// eDataMappingVarNames.powermonitor_events_b_EL3443Warning: 				st_Variable:= IotExtractType(monitor.powermonitor.events.b_EL3443Warning, 0, 0); 
// eDataMappingVarNames.powermonitor_events_b_EL3443Error: 				st_Variable:= IotExtractType(monitor.powermonitor.events.b_EL3443Error, 0, 0); 
// eDataMappingVarNames.powermonitor_events_b_ACdirectionDataInvalid: 				st_Variable:= IotExtractType(monitor.powermonitor.events.b_ACdirectionDataInvalid, 0, 0); 
// eDataMappingVarNames.ACswitchgear_b_InputSectionAvailable: 				st_Variable:= IotExtractType(monitor.ACswitchgear.b_InputSectionAvailable, 0, 0); 
// eDataMappingVarNames.ACswitchgear_b_InputMCCBfb: 				st_Variable:= IotExtractType(monitor.ACswitchgear.b_InputMCCBfb, 0, 0); 
// eDataMappingVarNames.ACswitchgear_b_InputMCCBShuntOK: 				st_Variable:= IotExtractType(monitor.ACswitchgear.b_InputMCCBShuntOK, 0, 0); 
// eDataMappingVarNames.ACswitchgear_b_OutputMCCBfb: 				st_Variable:= IotExtractType(monitor.ACswitchgear.b_OutputMCCBfb, 0, 0); 
// eDataMappingVarNames.ACswitchgear_b_OutputMCCBShuntOK: 				st_Variable:= IotExtractType(monitor.ACswitchgear.b_OutputMCCBShuntOK, 0, 0); 
// eDataMappingVarNames.ACswitchgear_b_CEEprefuseOK: 				st_Variable:= IotExtractType(monitor.ACswitchgear.b_CEEprefuseOK, 0, 0); 
// eDataMappingVarNames.ACswitchgear_b_InputSynchronizerfb: 				st_Variable:= IotExtractType(monitor.ACswitchgear.b_InputSynchronizerfb, 0, 0); 
// eDataMappingVarNames.ACswitchgear_b_InputContactorfb: 				st_Variable:= IotExtractType(monitor.ACswitchgear.b_InputContactorfb, 0, 0); 
// eDataMappingVarNames.ACswitchgear_b_PENlinkfb: 				st_Variable:= IotExtractType(monitor.ACswitchgear.b_PENlinkfb, 0, 0); 
// eDataMappingVarNames.ACswitchgear_events_b_InputMCCBShuntFault: 				st_Variable:= IotExtractType(monitor.ACswitchgear.events.b_InputMCCBShuntFault, 0, 0); 
// eDataMappingVarNames.ACswitchgear_events_b_OutputMCCBShuntFault: 				st_Variable:= IotExtractType(monitor.ACswitchgear.events.b_OutputMCCBShuntFault, 0, 0); 
// eDataMappingVarNames.ACswitchgear_events_b_CEEprefuseFault: 				st_Variable:= IotExtractType(monitor.ACswitchgear.events.b_CEEprefuseFault, 0, 0); 
// eDataMappingVarNames.ACswitchgear_events_b_InputContactorFault: 				st_Variable:= IotExtractType(monitor.ACswitchgear.events.b_InputContactorFault, 0, 0); 
// eDataMappingVarNames.neutraltransformer_b_active: 				st_Variable:= IotExtractType(monitor.neutraltransformer.b_active, 0, 0); 
// eDataMappingVarNames.neutraltransformer_r_TemperaturePhase_0: 				st_Variable:= IotExtractType(monitor.neutraltransformer.r_TemperaturePhase[0], 1, 0); 
// eDataMappingVarNames.neutraltransformer_r_TemperaturePhase_1: 				st_Variable:= IotExtractType(monitor.neutraltransformer.r_TemperaturePhase[1], 1, 0); 
// eDataMappingVarNames.neutraltransformer_r_TemperaturePhase_2: 				st_Variable:= IotExtractType(monitor.neutraltransformer.r_TemperaturePhase[2], 1, 0); 
// eDataMappingVarNames.neutraltransformer_r_TemperaturePhase_3: 				st_Variable:= IotExtractType(monitor.neutraltransformer.r_TemperaturePhase[3], 1, 0); 
// eDataMappingVarNames.neutraltransformer_r_TemperaturePhase_4: 				st_Variable:= IotExtractType(monitor.neutraltransformer.r_TemperaturePhase[4], 1, 0); 
// eDataMappingVarNames.neutraltransformer_r_TemperaturePhase_5: 				st_Variable:= IotExtractType(monitor.neutraltransformer.r_TemperaturePhase[5], 1, 0); 
// eDataMappingVarNames.neutraltransformer_r_TemperaturePhase_6: 				st_Variable:= IotExtractType(monitor.neutraltransformer.r_TemperaturePhase[6], 1, 0); 
// eDataMappingVarNames.neutraltransformer_r_Powerload: 				st_Variable:= IotExtractType(monitor.neutraltransformer.r_Powerload, 1, 0); 
// eDataMappingVarNames.neutraltransformer_r_ratedPower: 				st_Variable:= IotExtractType(monitor.neutraltransformer.r_ratedPower, 0, 0); 
// eDataMappingVarNames.neutraltransformer_events_b_TemperatureHighPhase_1: 				st_Variable:= IotExtractType(monitor.neutraltransformer.events.b_TemperatureHighPhase[1], 0, 0); 
// eDataMappingVarNames.neutraltransformer_events_b_TemperatureHighPhase_2: 				st_Variable:= IotExtractType(monitor.neutraltransformer.events.b_TemperatureHighPhase[2], 0, 0); 
// eDataMappingVarNames.neutraltransformer_events_b_TemperatureHighPhase_3: 				st_Variable:= IotExtractType(monitor.neutraltransformer.events.b_TemperatureHighPhase[3], 0, 0); 
// eDataMappingVarNames.neutraltransformer_events_b_TemperatureTooHighPhase_1: 				st_Variable:= IotExtractType(monitor.neutraltransformer.events.b_TemperatureTooHighPhase[1], 0, 0); 
// eDataMappingVarNames.neutraltransformer_events_b_TemperatureTooHighPhase_2: 				st_Variable:= IotExtractType(monitor.neutraltransformer.events.b_TemperatureTooHighPhase[2], 0, 0); 
// eDataMappingVarNames.neutraltransformer_events_b_TemperatureTooHighPhase_3: 				st_Variable:= IotExtractType(monitor.neutraltransformer.events.b_TemperatureTooHighPhase[3], 0, 0); 
// eDataMappingVarNames.neutraltransformer_events_b_VoltageUnbalanceHigh: 				st_Variable:= IotExtractType(monitor.neutraltransformer.events.b_VoltageUnbalanceHigh, 0, 0); 
// eDataMappingVarNames.neutraltransformer_events_b_VoltageUnbalanceTooHigh: 				st_Variable:= IotExtractType(monitor.neutraltransformer.events.b_VoltageUnbalanceTooHigh, 0, 0); 
// eDataMappingVarNames.neutraltransformer_events_b_NeutralCurrentHigh: 				st_Variable:= IotExtractType(monitor.neutraltransformer.events.b_NeutralCurrentHigh, 0, 0); 
// eDataMappingVarNames.neutraltransformer_events_b_NeutralCurrentTooHigh: 				st_Variable:= IotExtractType(monitor.neutraltransformer.events.b_NeutralCurrentTooHigh, 0, 0); 
// eDataMappingVarNames.neutraltransformer_events_b_OvercurrentWarning: 				st_Variable:= IotExtractType(monitor.neutraltransformer.events.b_OvercurrentWarning, 0, 0); 
// eDataMappingVarNames.neutraltransformer_events_b_OvercurrentAlarm: 				st_Variable:= IotExtractType(monitor.neutraltransformer.events.b_OvercurrentAlarm, 0, 0); 
// eDataMappingVarNames.DCswitchgear_b_CouplingState: 				st_Variable:= IotExtractType(monitor.DCswitchgear.b_CouplingState, 0, 0); 
// eDataMappingVarNames.DCswitchgear_r_Current: 				st_Variable:= IotExtractType(monitor.DCswitchgear.r_Current, 0, 0); 
// eDataMappingVarNames.DCswitchgear_r_ratedCurrent: 				st_Variable:= IotExtractType(monitor.DCswitchgear.r_ratedCurrent, 0, 0); 
// eDataMappingVarNames.battery_BatteryInfo_b_BMSHeartBeatOK: 				st_Variable:= IotExtractType(monitor.battery.BatteryInfo.b_BMSHeartBeatOK, 0, 0); 
// eDataMappingVarNames.battery_BatteryInfo_e_BMS_PowerOnStatus: 				st_Variable:= IotExtractType(monitor.battery.BatteryInfo.e_BMS_PowerOnStatus, 0, 0); 
// eDataMappingVarNames.battery_BatteryInfo_e_BMS_Status: 				st_Variable:= IotExtractType(monitor.battery.BatteryInfo.e_BMS_Status, 0, 0); 
// eDataMappingVarNames.battery_BatteryInfo_r_SystemVoltage: 				st_Variable:= IotExtractType(monitor.battery.BatteryInfo.r_SystemVoltage, 1, 0); 
// eDataMappingVarNames.battery_BatteryInfo_r_SystemCurrent: 				st_Variable:= IotExtractType(monitor.battery.BatteryInfo.r_SystemCurrent, 1, 0); 
// eDataMappingVarNames.battery_BatteryInfo_r_SOC: 				st_Variable:= IotExtractType(monitor.battery.BatteryInfo.r_SOC, 1, 0); 
// eDataMappingVarNames.battery_BatteryInfo_r_SOH: 				st_Variable:= IotExtractType(monitor.battery.BatteryInfo.r_SOH, 1, 0); 
// eDataMappingVarNames.battery_BatteryInfo_ar_CellVoltage_0: 				st_Variable:= IotExtractType(monitor.battery.BatteryInfo.ar_CellVoltage[0], 2, 0); 
// eDataMappingVarNames.battery_BatteryInfo_ar_CellVoltage_1: 				st_Variable:= IotExtractType(monitor.battery.BatteryInfo.ar_CellVoltage[1], 2, 0); 
// eDataMappingVarNames.battery_BatteryInfo_ar_CellVoltage_2: 				st_Variable:= IotExtractType(monitor.battery.BatteryInfo.ar_CellVoltage[2], 2, 0); 
// eDataMappingVarNames.battery_BatteryInfo_ar_CellTemperature_0: 				st_Variable:= IotExtractType(monitor.battery.BatteryInfo.ar_CellTemperature[0], 1, 0); 
// eDataMappingVarNames.battery_BatteryInfo_ar_CellTemperature_1: 				st_Variable:= IotExtractType(monitor.battery.BatteryInfo.ar_CellTemperature[1], 1, 0); 
// eDataMappingVarNames.battery_BatteryInfo_ar_CellTemperature_2: 				st_Variable:= IotExtractType(monitor.battery.BatteryInfo.ar_CellTemperature[2], 1, 0); 
// eDataMappingVarNames.battery_BatteryInfo_r_MaxChargeCurrentAllowed: 				st_Variable:= IotExtractType(monitor.battery.BatteryInfo.r_MaxChargeCurrentAllowed, 0, 0); 
// eDataMappingVarNames.battery_BatteryInfo_r_MaxDischargeCurrentAllowed: 				st_Variable:= IotExtractType(monitor.battery.BatteryInfo.r_MaxDischargeCurrentAllowed, 0, 0); 
// eDataMappingVarNames.battery_BatteryInfo_r_MaxChargePowerAllowed: 				st_Variable:= IotExtractType(monitor.battery.BatteryInfo.r_MaxChargePowerAllowed, 0, 0); 
// eDataMappingVarNames.battery_BatteryInfo_r_MaxDischargePowerAllowed: 				st_Variable:= IotExtractType(monitor.battery.BatteryInfo.r_MaxDischargePowerAllowed, 0, 0); 
// eDataMappingVarNames.battery_BatteryInfo_r_MaxSystemVoltageAllowed: 				st_Variable:= IotExtractType(monitor.battery.BatteryInfo.r_MaxSystemVoltageAllowed, 0, 0); 
// eDataMappingVarNames.battery_BatteryInfo_r_MinSystemVoltageAllowed: 				st_Variable:= IotExtractType(monitor.battery.BatteryInfo.r_MinSystemVoltageAllowed, 0, 0); 
// eDataMappingVarNames.battery_BatteryInfo_r_SystemPower: 				st_Variable:= IotExtractType(monitor.battery.BatteryInfo.r_SystemPower, 1, 0); 
// eDataMappingVarNames.battery_BatteryInfo_r_ChargeSOE: 				st_Variable:= IotExtractType(monitor.battery.BatteryInfo.r_ChargeSOE, 0, 0); 
// eDataMappingVarNames.battery_BatteryInfo_r_DischargeSOE: 				st_Variable:= IotExtractType(monitor.battery.BatteryInfo.r_DischargeSOE, 0, 0); 
// eDataMappingVarNames.battery_BatteryInfo_r_RemainingChargeEnergy: 				st_Variable:= IotExtractType(monitor.battery.BatteryInfo.r_RemainingChargeEnergy, 0, 0); 
// eDataMappingVarNames.battery_BatteryInfo_r_RemainingDischargeEnergy: 				st_Variable:= IotExtractType(monitor.battery.BatteryInfo.r_RemainingDischargeEnergy, 0, 0); 
// eDataMappingVarNames.battery_BatteryInfo_r_HistAccChargeEnergy: 				st_Variable:= IotExtractType(monitor.battery.BatteryInfo.r_HistAccChargeEnergy, 0, 0); 
// eDataMappingVarNames.battery_BatteryInfo_r_HistAccDischargeEnergy: 				st_Variable:= IotExtractType(monitor.battery.BatteryInfo.r_HistAccDischargeEnergy, 0, 0); 
// eDataMappingVarNames.battery_BatteryInfo_r_ratedPower: 				st_Variable:= IotExtractType(monitor.battery.BatteryInfo.r_ratedPower, 0, 0); 
// eDataMappingVarNames.battery_BatteryInfo_r_ratedCurrent: 				st_Variable:= IotExtractType(monitor.battery.BatteryInfo.r_ratedCurrent, 0, 0); 
// eDataMappingVarNames.battery_BatteryInfo_r_ratedEnergyCapacity: 				st_Variable:= IotExtractType(monitor.battery.BatteryInfo.r_ratedEnergyCapacity, 0, 0); 
// eDataMappingVarNames.battery_BatteryInfo_ui_CycleCount: 				st_Variable:= IotExtractType(monitor.battery.BatteryInfo.ui_CycleCount, 0, 0); 
// eDataMappingVarNames.battery_BatteryInfo_r_SOCScaled: 				st_Variable:= IotExtractType(monitor.battery.BatteryInfo.r_SOCScaled, 1, 0); 
// eDataMappingVarNames.battery_BatteryInfo_b_chargingAllowed: 				st_Variable:= IotExtractType(monitor.battery.BatteryInfo.b_chargingAllowed, 0, 0); 
// eDataMappingVarNames.battery_BatteryInfo_b_dischargingAllowed: 				st_Variable:= IotExtractType(monitor.battery.BatteryInfo.b_dischargingAllowed, 0, 0); 
// eDataMappingVarNames.battery_BatteryInfo_r_RemainingDischargeEnergyNett: 				st_Variable:= IotExtractType(monitor.battery.BatteryInfo.r_RemainingDischargeEnergyNett, 0, 0); 
// eDataMappingVarNames.battery_BatteryInfo_r_RemainingChargeEnergyNett: 				st_Variable:= IotExtractType(monitor.battery.BatteryInfo.r_RemainingChargeEnergyNett, 0, 0); 
// eDataMappingVarNames.battery_BatteryInfo_r_maxVoltageEver: 				st_Variable:= IotExtractType(monitor.battery.BatteryInfo.r_maxVoltageEver, 1, 0); 
// eDataMappingVarNames.battery_BatteryInfo_r_maxChargeCurrentEver: 				st_Variable:= IotExtractType(monitor.battery.BatteryInfo.r_maxChargeCurrentEver, 1, 0); 
// eDataMappingVarNames.battery_BatteryInfo_r_maxDischargeCurrentEver: 				st_Variable:= IotExtractType(monitor.battery.BatteryInfo.r_maxDischargeCurrentEver, 1, 0); 
// eDataMappingVarNames.battery_T_RemainingTimeToAutoCalibration: 				st_Variable:= IotExtractType(monitor.battery.T_RemainingTimeToAutoCalibration, 0, 0); 
// eDataMappingVarNames.battery_MBMU_GeneralSBMUStatus_0: 				st_Variable:= IotExtractType(monitor.battery.MBMU.GeneralSBMUStatus[0], 0, 0); 
// eDataMappingVarNames.battery_MBMU_GeneralSBMUStatus_1: 				st_Variable:= IotExtractType(monitor.battery.MBMU.GeneralSBMUStatus[1], 0, 0); 
// eDataMappingVarNames.battery_MBMU_GeneralSBMUStatus_2: 				st_Variable:= IotExtractType(monitor.battery.MBMU.GeneralSBMUStatus[2], 0, 0); 
// eDataMappingVarNames.battery_MBMU_GeneralSBMUStatus_3: 				st_Variable:= IotExtractType(monitor.battery.MBMU.GeneralSBMUStatus[3], 0, 0); 
// eDataMappingVarNames.battery_MBMU_GeneralSBMUStatus_4: 				st_Variable:= IotExtractType(monitor.battery.MBMU.GeneralSBMUStatus[4], 0, 0); 
// eDataMappingVarNames.battery_MBMU_GeneralSBMUStatus_5: 				st_Variable:= IotExtractType(monitor.battery.MBMU.GeneralSBMUStatus[5], 0, 0); 
// eDataMappingVarNames.battery_MBMU_GeneralSBMUStatus_6: 				st_Variable:= IotExtractType(monitor.battery.MBMU.GeneralSBMUStatus[6], 0, 0); 
// eDataMappingVarNames.battery_MBMU_GeneralSBMUStatus_7: 				st_Variable:= IotExtractType(monitor.battery.MBMU.GeneralSBMUStatus[7], 0, 0); 
// eDataMappingVarNames.battery_MBMU_GeneralSBMUStatus_8: 				st_Variable:= IotExtractType(monitor.battery.MBMU.GeneralSBMUStatus[8], 0, 0); 
// eDataMappingVarNames.battery_MBMU_GeneralSBMUStatus_9: 				st_Variable:= IotExtractType(monitor.battery.MBMU.GeneralSBMUStatus[9], 0, 0); 
// eDataMappingVarNames.battery_MBMU_GeneralSBMUStatus_10: 				st_Variable:= IotExtractType(monitor.battery.MBMU.GeneralSBMUStatus[10], 0, 0); 
// eDataMappingVarNames.battery_MBMU_GeneralSBMUStatus_11: 				st_Variable:= IotExtractType(monitor.battery.MBMU.GeneralSBMUStatus[11], 0, 0); 
// eDataMappingVarNames.battery_MBMU_GeneralSBMUStatus_12: 				st_Variable:= IotExtractType(monitor.battery.MBMU.GeneralSBMUStatus[12], 0, 0); 
// eDataMappingVarNames.battery_MBMU_GeneralSBMUStatus_13: 				st_Variable:= IotExtractType(monitor.battery.MBMU.GeneralSBMUStatus[13], 0, 0); 
// eDataMappingVarNames.battery_MBMU_GeneralSBMUStatus_14: 				st_Variable:= IotExtractType(monitor.battery.MBMU.GeneralSBMUStatus[14], 0, 0); 
// eDataMappingVarNames.battery_MBMU_GeneralSBMUStatus_15: 				st_Variable:= IotExtractType(monitor.battery.MBMU.GeneralSBMUStatus[15], 0, 0); 
// eDataMappingVarNames.battery_MBMU_MBMUStatus_0: 				st_Variable:= IotExtractType(monitor.battery.MBMU.MBMUStatus[0], 0, 0); 
// eDataMappingVarNames.battery_MBMU_MBMUStatus_1: 				st_Variable:= IotExtractType(monitor.battery.MBMU.MBMUStatus[1], 0, 0); 
// eDataMappingVarNames.battery_MBMU_MBMUStatus_2: 				st_Variable:= IotExtractType(monitor.battery.MBMU.MBMUStatus[2], 0, 0); 
// eDataMappingVarNames.battery_MBMU_MBMUStatus_3: 				st_Variable:= IotExtractType(monitor.battery.MBMU.MBMUStatus[3], 0, 0); 
// eDataMappingVarNames.battery_MBMU_MBMUStatus_4: 				st_Variable:= IotExtractType(monitor.battery.MBMU.MBMUStatus[4], 0, 0); 
// eDataMappingVarNames.battery_MBMU_MBMUStatus_5: 				st_Variable:= IotExtractType(monitor.battery.MBMU.MBMUStatus[5], 0, 0); 
// eDataMappingVarNames.battery_MBMU_MBMUStatus_6: 				st_Variable:= IotExtractType(monitor.battery.MBMU.MBMUStatus[6], 0, 0); 
// eDataMappingVarNames.battery_MBMU_MBMUStatus_7: 				st_Variable:= IotExtractType(monitor.battery.MBMU.MBMUStatus[7], 0, 0); 
// eDataMappingVarNames.battery_MBMU_MBMUStatus_8: 				st_Variable:= IotExtractType(monitor.battery.MBMU.MBMUStatus[8], 0, 0); 
// eDataMappingVarNames.battery_MBMU_MBMUStatus_9: 				st_Variable:= IotExtractType(monitor.battery.MBMU.MBMUStatus[9], 0, 0); 
// eDataMappingVarNames.battery_MBMU_MBMUStatus_10: 				st_Variable:= IotExtractType(monitor.battery.MBMU.MBMUStatus[10], 0, 0); 
// eDataMappingVarNames.battery_MBMU_MBMUStatus_11: 				st_Variable:= IotExtractType(monitor.battery.MBMU.MBMUStatus[11], 0, 0); 
// eDataMappingVarNames.battery_MBMU_MBMUStatus_12: 				st_Variable:= IotExtractType(monitor.battery.MBMU.MBMUStatus[12], 0, 0); 
// eDataMappingVarNames.battery_MBMU_MBMUStatus_13: 				st_Variable:= IotExtractType(monitor.battery.MBMU.MBMUStatus[13], 0, 0); 
// eDataMappingVarNames.battery_MBMU_MBMUStatus_14: 				st_Variable:= IotExtractType(monitor.battery.MBMU.MBMUStatus[14], 0, 0); 
// eDataMappingVarNames.battery_MBMU_MBMUStatus_15: 				st_Variable:= IotExtractType(monitor.battery.MBMU.MBMUStatus[15], 0, 0); 
// eDataMappingVarNames.battery_MBMU_s_MBMU_SWVer: 				st_Variable:= IotExtractType(monitor.battery.MBMU.s_MBMU_SWVer, 0, 0); 
// eDataMappingVarNames.battery_MBMU_s_MBMU_HWVer: 				st_Variable:= IotExtractType(monitor.battery.MBMU.s_MBMU_HWVer, 0, 0); 
// eDataMappingVarNames.battery_MBMU_s_ETH_SWVer: 				st_Variable:= IotExtractType(monitor.battery.MBMU.s_ETH_SWVer, 0, 0); 
// eDataMappingVarNames.battery_MBMU_r_ETH_HWVer: 				st_Variable:= IotExtractType(monitor.battery.MBMU.r_ETH_HWVer, 0, 0); 
// eDataMappingVarNames.battery_MBMU_by_NumberOfSubSystems: 				st_Variable:= IotExtractType(monitor.battery.MBMU.by_NumberOfSubSystems, 0, 0); 
// eDataMappingVarNames.battery_MBMU_DateTime_0: 				st_Variable:= IotExtractType(monitor.battery.MBMU.DateTime[0], 0, 0); 
// eDataMappingVarNames.battery_MBMU_DateTime_1: 				st_Variable:= IotExtractType(monitor.battery.MBMU.DateTime[1], 0, 0); 
// eDataMappingVarNames.battery_MBMU_DateTime_2: 				st_Variable:= IotExtractType(monitor.battery.MBMU.DateTime[2], 0, 0); 
// eDataMappingVarNames.battery_MBMU_DateTime_3: 				st_Variable:= IotExtractType(monitor.battery.MBMU.DateTime[3], 0, 0); 
// eDataMappingVarNames.battery_MBMU_DateTime_4: 				st_Variable:= IotExtractType(monitor.battery.MBMU.DateTime[4], 0, 0); 
// eDataMappingVarNames.battery_MBMU_DateTime_5: 				st_Variable:= IotExtractType(monitor.battery.MBMU.DateTime[5], 0, 0); 
// eDataMappingVarNames.battery_MBMU_b_InsulationSwitchOpen: 				st_Variable:= IotExtractType(monitor.battery.MBMU.b_InsulationSwitchOpen, 0, 0); 
// eDataMappingVarNames.battery_MBMU_BatteryStatus_b_BMSHeartBeatOK: 				st_Variable:= IotExtractType(monitor.battery.MBMU.BatteryStatus.b_BMSHeartBeatOK, 0, 0); 
// eDataMappingVarNames.battery_MBMU_BatteryStatus_e_BMS_PowerOnStatus: 				st_Variable:= IotExtractType(monitor.battery.MBMU.BatteryStatus.e_BMS_PowerOnStatus, 0, 0); 
// eDataMappingVarNames.battery_MBMU_BatteryStatus_e_BMS_Status: 					st_Variable:= IotExtractType(monitor.battery.MBMU.BatteryStatus.e_BMS_Status, 0, 0); 
// eDataMappingVarNames.battery_MBMU_BatteryStatus_r_SystemVoltage: 				st_Variable:= IotExtractType(monitor.battery.MBMU.BatteryStatus.r_SystemVoltage, 0, 0); 
// eDataMappingVarNames.battery_MBMU_BatteryStatus_r_SystemCurrent: 				st_Variable:= IotExtractType(monitor.battery.MBMU.BatteryStatus.r_SystemCurrent, 0, 0); 
// eDataMappingVarNames.battery_MBMU_BatteryStatus_r_SOC: 							st_Variable:= IotExtractType(monitor.battery.MBMU.BatteryStatus.r_SOC, 1, 0); 
// eDataMappingVarNames.battery_MBMU_BatteryStatus_r_SOH: 							st_Variable:= IotExtractType(monitor.battery.MBMU.BatteryStatus.r_SOH, 1, 0); 
// eDataMappingVarNames.battery_MBMU_BatteryStatus_ar_CellVoltage_0: 				st_Variable:= IotExtractType(monitor.battery.MBMU.BatteryStatus.ar_CellVoltage[0], 2, 0); 
// eDataMappingVarNames.battery_MBMU_BatteryStatus_ar_CellVoltage_1: 				st_Variable:= IotExtractType(monitor.battery.MBMU.BatteryStatus.ar_CellVoltage[1], 2, 0); 
// eDataMappingVarNames.battery_MBMU_BatteryStatus_ar_CellVoltage_2: 				st_Variable:= IotExtractType(monitor.battery.MBMU.BatteryStatus.ar_CellVoltage[2], 2, 0); 
// eDataMappingVarNames.battery_MBMU_BatteryStatus_ar_CellTemperature_0: 				st_Variable:= IotExtractType(monitor.battery.MBMU.BatteryStatus.ar_CellTemperature[0], 1, 0); 
// eDataMappingVarNames.battery_MBMU_BatteryStatus_ar_CellTemperature_1: 				st_Variable:= IotExtractType(monitor.battery.MBMU.BatteryStatus.ar_CellTemperature[1], 1, 0); 
// eDataMappingVarNames.battery_MBMU_BatteryStatus_ar_CellTemperature_2: 				st_Variable:= IotExtractType(monitor.battery.MBMU.BatteryStatus.ar_CellTemperature[2], 1, 0); 
// eDataMappingVarNames.battery_MBMU_BatteryStatus_r_MaxChargeCurrentAllowed: 				st_Variable:= IotExtractType(monitor.battery.MBMU.BatteryStatus.r_MaxChargeCurrentAllowed, 0, 0); 
// eDataMappingVarNames.battery_MBMU_BatteryStatus_r_MaxDischargeCurrentAllowed: 				st_Variable:= IotExtractType(monitor.battery.MBMU.BatteryStatus.r_MaxDischargeCurrentAllowed, 0, 0); 
// eDataMappingVarNames.battery_MBMU_BatteryStatus_r_MaxChargePowerAllowed: 				st_Variable:= IotExtractType(monitor.battery.MBMU.BatteryStatus.r_MaxChargePowerAllowed, 0, 0); 
// eDataMappingVarNames.battery_MBMU_BatteryStatus_r_MaxDischargePowerAllowed: 				st_Variable:= IotExtractType(monitor.battery.MBMU.BatteryStatus.r_MaxDischargePowerAllowed, 0, 0); 
// eDataMappingVarNames.battery_MBMU_BatteryStatus_r_MaxSystemVoltageAllowed: 				st_Variable:= IotExtractType(monitor.battery.MBMU.BatteryStatus.r_MaxSystemVoltageAllowed, 0, 0); 
// eDataMappingVarNames.battery_MBMU_BatteryStatus_r_MinSystemVoltageAllowed: 				st_Variable:= IotExtractType(monitor.battery.MBMU.BatteryStatus.r_MinSystemVoltageAllowed, 0, 0); 
// eDataMappingVarNames.battery_MBMU_BatteryStatus_r_SystemPower: 				st_Variable:= IotExtractType(monitor.battery.MBMU.BatteryStatus.r_SystemPower, 1, 0); 
// eDataMappingVarNames.battery_MBMU_BatteryStatus_r_ChargeSOE: 				st_Variable:= IotExtractType(monitor.battery.MBMU.BatteryStatus.r_ChargeSOE, 0, 0); 
// eDataMappingVarNames.battery_MBMU_BatteryStatus_r_DischargeSOE: 				st_Variable:= IotExtractType(monitor.battery.MBMU.BatteryStatus.r_DischargeSOE, 0, 0); 
// eDataMappingVarNames.battery_MBMU_BatteryStatus_r_RemainingChargeEnergy: 				st_Variable:= IotExtractType(monitor.battery.MBMU.BatteryStatus.r_RemainingChargeEnergy, 0, 0); 
// eDataMappingVarNames.battery_MBMU_BatteryStatus_r_RemainingDischargeEnergy: 				st_Variable:= IotExtractType(monitor.battery.MBMU.BatteryStatus.r_RemainingDischargeEnergy, 0, 0); 
// eDataMappingVarNames.battery_MBMU_BatteryStatus_r_HistAccChargeEnergy: 				st_Variable:= IotExtractType(monitor.battery.MBMU.BatteryStatus.r_HistAccChargeEnergy, 0, 0); 
// eDataMappingVarNames.battery_MBMU_BatteryStatus_r_HistAccDischargeEnergy: 				st_Variable:= IotExtractType(monitor.battery.MBMU.BatteryStatus.r_HistAccDischargeEnergy, 0, 0); 
// eDataMappingVarNames.battery_SBMU_0_w_SystemWarning: 				st_Variable:= IotExtractType(monitor.battery.SBMU[0].w_SystemWarning, 0, 0); 
// eDataMappingVarNames.battery_SBMU_1_w_SystemWarning: 				st_Variable:= IotExtractType(monitor.battery.SBMU[1].w_SystemWarning, 0, 0); 
// eDataMappingVarNames.battery_SBMU_2_w_SystemWarning: 				st_Variable:= IotExtractType(monitor.battery.SBMU[2].w_SystemWarning, 0, 0); 
// eDataMappingVarNames.battery_SBMU_3_w_SystemWarning: 				st_Variable:= IotExtractType(monitor.battery.SBMU[3].w_SystemWarning, 0, 0); 
// eDataMappingVarNames.battery_SBMU_0_SystemAlarm_0: 				st_Variable:= IotExtractType(monitor.battery.SBMU[0].SystemAlarm[0], 0, 0); 
// eDataMappingVarNames.battery_SBMU_1_SystemAlarm_0: 				st_Variable:= IotExtractType(monitor.battery.SBMU[1].SystemAlarm[0], 0, 0); 
// eDataMappingVarNames.battery_SBMU_2_SystemAlarm_0: 				st_Variable:= IotExtractType(monitor.battery.SBMU[2].SystemAlarm[0], 0, 0); 
// eDataMappingVarNames.battery_SBMU_3_SystemAlarm_0: 				st_Variable:= IotExtractType(monitor.battery.SBMU[3].SystemAlarm[0], 0, 0); 
// eDataMappingVarNames.battery_SBMU_0_SystemAlarm_1: 				st_Variable:= IotExtractType(monitor.battery.SBMU[0].SystemAlarm[1], 0, 0); 
// eDataMappingVarNames.battery_SBMU_1_SystemAlarm_1: 				st_Variable:= IotExtractType(monitor.battery.SBMU[1].SystemAlarm[1], 0, 0); 
// eDataMappingVarNames.battery_SBMU_2_SystemAlarm_1: 				st_Variable:= IotExtractType(monitor.battery.SBMU[2].SystemAlarm[1], 0, 0); 
// eDataMappingVarNames.battery_SBMU_3_SystemAlarm_1: 				st_Variable:= IotExtractType(monitor.battery.SBMU[3].SystemAlarm[1], 0, 0); 
// eDataMappingVarNames.battery_SBMU_0_SystemAlarm_2: 				st_Variable:= IotExtractType(monitor.battery.SBMU[0].SystemAlarm[2], 0, 0); 
// eDataMappingVarNames.battery_SBMU_1_SystemAlarm_2: 				st_Variable:= IotExtractType(monitor.battery.SBMU[1].SystemAlarm[2], 0, 0); 
// eDataMappingVarNames.battery_SBMU_2_SystemAlarm_2: 				st_Variable:= IotExtractType(monitor.battery.SBMU[2].SystemAlarm[2], 0, 0); 
// eDataMappingVarNames.battery_SBMU_3_SystemAlarm_2: 				st_Variable:= IotExtractType(monitor.battery.SBMU[3].SystemAlarm[2], 0, 0); 
// eDataMappingVarNames.battery_SBMU_0_b_PrechargeRelayClosed: 				st_Variable:= IotExtractType(monitor.battery.SBMU[0].b_PrechargeRelayClosed, 0, 0); 
// eDataMappingVarNames.battery_SBMU_1_b_PrechargeRelayClosed: 				st_Variable:= IotExtractType(monitor.battery.SBMU[1].b_PrechargeRelayClosed, 0, 0); 
// eDataMappingVarNames.battery_SBMU_2_b_PrechargeRelayClosed: 				st_Variable:= IotExtractType(monitor.battery.SBMU[2].b_PrechargeRelayClosed, 0, 0); 
// eDataMappingVarNames.battery_SBMU_3_b_PrechargeRelayClosed: 				st_Variable:= IotExtractType(monitor.battery.SBMU[3].b_PrechargeRelayClosed, 0, 0); 
// eDataMappingVarNames.battery_SBMU_0_b_MainPosRelayClosed: 				st_Variable:= IotExtractType(monitor.battery.SBMU[0].b_MainPosRelayClosed, 0, 0); 
// eDataMappingVarNames.battery_SBMU_1_b_MainPosRelayClosed: 				st_Variable:= IotExtractType(monitor.battery.SBMU[1].b_MainPosRelayClosed, 0, 0); 
// eDataMappingVarNames.battery_SBMU_2_b_MainPosRelayClosed: 				st_Variable:= IotExtractType(monitor.battery.SBMU[2].b_MainPosRelayClosed, 0, 0); 
// eDataMappingVarNames.battery_SBMU_3_b_MainPosRelayClosed: 				st_Variable:= IotExtractType(monitor.battery.SBMU[3].b_MainPosRelayClosed, 0, 0); 
// eDataMappingVarNames.battery_SBMU_0_b_MainNegRelayClosed: 				st_Variable:= IotExtractType(monitor.battery.SBMU[0].b_MainNegRelayClosed, 0, 0); 
// eDataMappingVarNames.battery_SBMU_1_b_MainNegRelayClosed: 				st_Variable:= IotExtractType(monitor.battery.SBMU[1].b_MainNegRelayClosed, 0, 0); 
// eDataMappingVarNames.battery_SBMU_2_b_MainNegRelayClosed: 				st_Variable:= IotExtractType(monitor.battery.SBMU[2].b_MainNegRelayClosed, 0, 0); 
// eDataMappingVarNames.battery_SBMU_3_b_MainNegRelayClosed: 				st_Variable:= IotExtractType(monitor.battery.SBMU[3].b_MainNegRelayClosed, 0, 0); 
// eDataMappingVarNames.battery_SBMU_0_b_ControlBoxFanOn: 				st_Variable:= IotExtractType(monitor.battery.SBMU[0].b_ControlBoxFanOn, 0, 0); 
// eDataMappingVarNames.battery_SBMU_1_b_ControlBoxFanOn: 				st_Variable:= IotExtractType(monitor.battery.SBMU[1].b_ControlBoxFanOn, 0, 0); 
// eDataMappingVarNames.battery_SBMU_2_b_ControlBoxFanOn: 				st_Variable:= IotExtractType(monitor.battery.SBMU[2].b_ControlBoxFanOn, 0, 0); 
// eDataMappingVarNames.battery_SBMU_3_b_ControlBoxFanOn: 				st_Variable:= IotExtractType(monitor.battery.SBMU[3].b_ControlBoxFanOn, 0, 0); 
// eDataMappingVarNames.battery_SBMU_0_b_BalanceStatus: 				st_Variable:= IotExtractType(monitor.battery.SBMU[0].b_BalanceStatus, 0, 0); 
// eDataMappingVarNames.battery_SBMU_1_b_BalanceStatus: 				st_Variable:= IotExtractType(monitor.battery.SBMU[1].b_BalanceStatus, 0, 0); 
// eDataMappingVarNames.battery_SBMU_2_b_BalanceStatus: 				st_Variable:= IotExtractType(monitor.battery.SBMU[2].b_BalanceStatus, 0, 0); 
// eDataMappingVarNames.battery_SBMU_3_b_BalanceStatus: 				st_Variable:= IotExtractType(monitor.battery.SBMU[3].b_BalanceStatus, 0, 0); 
// eDataMappingVarNames.battery_SBMU_0_b_DoorState: 				st_Variable:= IotExtractType(monitor.battery.SBMU[0].b_DoorState, 0, 0); 
// eDataMappingVarNames.battery_SBMU_1_b_DoorState: 				st_Variable:= IotExtractType(monitor.battery.SBMU[1].b_DoorState, 0, 0); 
// eDataMappingVarNames.battery_SBMU_2_b_DoorState: 				st_Variable:= IotExtractType(monitor.battery.SBMU[2].b_DoorState, 0, 0); 
// eDataMappingVarNames.battery_SBMU_3_b_DoorState: 				st_Variable:= IotExtractType(monitor.battery.SBMU[3].b_DoorState, 0, 0); 
// eDataMappingVarNames.battery_SBMU_0_s_SBMU_SWVer: 				st_Variable:= IotExtractType(monitor.battery.SBMU[0].s_SBMU_SWVer, 0, 0); 
// eDataMappingVarNames.battery_SBMU_1_s_SBMU_SWVer: 				st_Variable:= IotExtractType(monitor.battery.SBMU[1].s_SBMU_SWVer, 0, 0); 
// eDataMappingVarNames.battery_SBMU_2_s_SBMU_SWVer: 				st_Variable:= IotExtractType(monitor.battery.SBMU[2].s_SBMU_SWVer, 0, 0); 
// eDataMappingVarNames.battery_SBMU_3_s_SBMU_SWVer: 				st_Variable:= IotExtractType(monitor.battery.SBMU[3].s_SBMU_SWVer, 0, 0); 
// eDataMappingVarNames.battery_SBMU_0_s_SBMU_HWVer: 				st_Variable:= IotExtractType(monitor.battery.SBMU[0].s_SBMU_HWVer, 0, 0); 
// eDataMappingVarNames.battery_SBMU_1_s_SBMU_HWVer: 				st_Variable:= IotExtractType(monitor.battery.SBMU[1].s_SBMU_HWVer, 0, 0); 
// eDataMappingVarNames.battery_SBMU_2_s_SBMU_HWVer: 				st_Variable:= IotExtractType(monitor.battery.SBMU[2].s_SBMU_HWVer, 0, 0); 
// eDataMappingVarNames.battery_SBMU_3_s_SBMU_HWVer: 				st_Variable:= IotExtractType(monitor.battery.SBMU[3].s_SBMU_HWVer, 0, 0); 
// eDataMappingVarNames.battery_SBMU_0_s_CSC_SWVer: 				st_Variable:= IotExtractType(monitor.battery.SBMU[0].s_CSC_SWVer, 0, 0); 
// eDataMappingVarNames.battery_SBMU_1_s_CSC_SWVer: 				st_Variable:= IotExtractType(monitor.battery.SBMU[1].s_CSC_SWVer, 0, 0); 
// eDataMappingVarNames.battery_SBMU_2_s_CSC_SWVer: 				st_Variable:= IotExtractType(monitor.battery.SBMU[2].s_CSC_SWVer, 0, 0); 
// eDataMappingVarNames.battery_SBMU_3_s_CSC_SWVer: 				st_Variable:= IotExtractType(monitor.battery.SBMU[3].s_CSC_SWVer, 0, 0); 
// eDataMappingVarNames.battery_SBMU_0_s_CSC_HWVer: 				st_Variable:= IotExtractType(monitor.battery.SBMU[0].s_CSC_HWVer, 0, 0); 
// eDataMappingVarNames.battery_SBMU_1_s_CSC_HWVer: 				st_Variable:= IotExtractType(monitor.battery.SBMU[1].s_CSC_HWVer, 0, 0); 
// eDataMappingVarNames.battery_SBMU_2_s_CSC_HWVer: 				st_Variable:= IotExtractType(monitor.battery.SBMU[2].s_CSC_HWVer, 0, 0); 
// eDataMappingVarNames.battery_SBMU_3_s_CSC_HWVer: 				st_Variable:= IotExtractType(monitor.battery.SBMU[3].s_CSC_HWVer, 0, 0); 
// eDataMappingVarNames.battery_SBMU_0_BatteryStatus_r_SystemVoltage: 				st_Variable:= IotExtractType(monitor.battery.SBMU[0].BatteryStatus.r_SystemVoltage, 1, 0); 
// eDataMappingVarNames.battery_SBMU_1_BatteryStatus_r_SystemVoltage: 				st_Variable:= IotExtractType(monitor.battery.SBMU[1].BatteryStatus.r_SystemVoltage, 1, 0); 
// eDataMappingVarNames.battery_SBMU_2_BatteryStatus_r_SystemVoltage: 				st_Variable:= IotExtractType(monitor.battery.SBMU[2].BatteryStatus.r_SystemVoltage, 1, 0); 
// eDataMappingVarNames.battery_SBMU_3_BatteryStatus_r_SystemVoltage: 				st_Variable:= IotExtractType(monitor.battery.SBMU[3].BatteryStatus.r_SystemVoltage, 1, 0); 
// eDataMappingVarNames.battery_SBMU_0_BatteryStatus_r_SystemCurrent: 				st_Variable:= IotExtractType(monitor.battery.SBMU[0].BatteryStatus.r_SystemCurrent, 1, 0); 
// eDataMappingVarNames.battery_SBMU_1_BatteryStatus_r_SystemCurrent: 				st_Variable:= IotExtractType(monitor.battery.SBMU[1].BatteryStatus.r_SystemCurrent, 1, 0); 
// eDataMappingVarNames.battery_SBMU_2_BatteryStatus_r_SystemCurrent: 				st_Variable:= IotExtractType(monitor.battery.SBMU[2].BatteryStatus.r_SystemCurrent, 1, 0); 
// eDataMappingVarNames.battery_SBMU_3_BatteryStatus_r_SystemCurrent: 				st_Variable:= IotExtractType(monitor.battery.SBMU[3].BatteryStatus.r_SystemCurrent, 1, 0); 
// eDataMappingVarNames.battery_SBMU_0_BatteryStatus_r_SOC: 				st_Variable:= IotExtractType(monitor.battery.SBMU[0].BatteryStatus.r_SOC, 1, 0); 
// eDataMappingVarNames.battery_SBMU_1_BatteryStatus_r_SOC: 				st_Variable:= IotExtractType(monitor.battery.SBMU[1].BatteryStatus.r_SOC, 1, 0); 
// eDataMappingVarNames.battery_SBMU_2_BatteryStatus_r_SOC: 				st_Variable:= IotExtractType(monitor.battery.SBMU[2].BatteryStatus.r_SOC, 1, 0); 
// eDataMappingVarNames.battery_SBMU_3_BatteryStatus_r_SOC: 				st_Variable:= IotExtractType(monitor.battery.SBMU[3].BatteryStatus.r_SOC, 1, 0); 
// eDataMappingVarNames.battery_SBMU_0_BatteryStatus_r_SOH: 				st_Variable:= IotExtractType(monitor.battery.SBMU[0].BatteryStatus.r_SOH, 1, 0); 
// eDataMappingVarNames.battery_SBMU_1_BatteryStatus_r_SOH: 				st_Variable:= IotExtractType(monitor.battery.SBMU[1].BatteryStatus.r_SOH, 1, 0); 
// eDataMappingVarNames.battery_SBMU_2_BatteryStatus_r_SOH: 				st_Variable:= IotExtractType(monitor.battery.SBMU[2].BatteryStatus.r_SOH, 1, 0); 
// eDataMappingVarNames.battery_SBMU_3_BatteryStatus_r_SOH: 				st_Variable:= IotExtractType(monitor.battery.SBMU[3].BatteryStatus.r_SOH, 1, 0); 
// eDataMappingVarNames.battery_SBMU_0_BatteryStatus_ar_CellVoltage_0: 				st_Variable:= IotExtractType(monitor.battery.SBMU[0].BatteryStatus.ar_CellVoltage[0], 2, 0); 
// eDataMappingVarNames.battery_SBMU_1_BatteryStatus_ar_CellVoltage_0: 				st_Variable:= IotExtractType(monitor.battery.SBMU[1].BatteryStatus.ar_CellVoltage[0], 2, 0); 
// eDataMappingVarNames.battery_SBMU_2_BatteryStatus_ar_CellVoltage_0: 				st_Variable:= IotExtractType(monitor.battery.SBMU[2].BatteryStatus.ar_CellVoltage[0], 2, 0); 
// eDataMappingVarNames.battery_SBMU_3_BatteryStatus_ar_CellVoltage_0: 				st_Variable:= IotExtractType(monitor.battery.SBMU[3].BatteryStatus.ar_CellVoltage[0], 2, 0); 
// eDataMappingVarNames.battery_SBMU_0_BatteryStatus_ar_CellVoltage_1: 				st_Variable:= IotExtractType(monitor.battery.SBMU[0].BatteryStatus.ar_CellVoltage[1], 2, 0); 
// eDataMappingVarNames.battery_SBMU_1_BatteryStatus_ar_CellVoltage_1: 				st_Variable:= IotExtractType(monitor.battery.SBMU[1].BatteryStatus.ar_CellVoltage[1], 2, 0); 
// eDataMappingVarNames.battery_SBMU_2_BatteryStatus_ar_CellVoltage_1: 				st_Variable:= IotExtractType(monitor.battery.SBMU[2].BatteryStatus.ar_CellVoltage[1], 2, 0); 
// eDataMappingVarNames.battery_SBMU_3_BatteryStatus_ar_CellVoltage_1: 				st_Variable:= IotExtractType(monitor.battery.SBMU[3].BatteryStatus.ar_CellVoltage[1], 2, 0); 
// eDataMappingVarNames.battery_SBMU_0_BatteryStatus_ar_CellVoltage_2: 				st_Variable:= IotExtractType(monitor.battery.SBMU[0].BatteryStatus.ar_CellVoltage[2], 2, 0); 
// eDataMappingVarNames.battery_SBMU_1_BatteryStatus_ar_CellVoltage_2: 				st_Variable:= IotExtractType(monitor.battery.SBMU[1].BatteryStatus.ar_CellVoltage[2], 2, 0); 
// eDataMappingVarNames.battery_SBMU_2_BatteryStatus_ar_CellVoltage_2: 				st_Variable:= IotExtractType(monitor.battery.SBMU[2].BatteryStatus.ar_CellVoltage[2], 2, 0); 
// eDataMappingVarNames.battery_SBMU_3_BatteryStatus_ar_CellVoltage_2: 				st_Variable:= IotExtractType(monitor.battery.SBMU[3].BatteryStatus.ar_CellVoltage[2], 2, 0); 
// eDataMappingVarNames.battery_SBMU_0_BatteryStatus_ar_CellTemperature_0: 				st_Variable:= IotExtractType(monitor.battery.SBMU[0].BatteryStatus.ar_CellTemperature[0], 1, 0); 
// eDataMappingVarNames.battery_SBMU_1_BatteryStatus_ar_CellTemperature_0: 				st_Variable:= IotExtractType(monitor.battery.SBMU[1].BatteryStatus.ar_CellTemperature[0], 1, 0); 
// eDataMappingVarNames.battery_SBMU_2_BatteryStatus_ar_CellTemperature_0: 				st_Variable:= IotExtractType(monitor.battery.SBMU[2].BatteryStatus.ar_CellTemperature[0], 1, 0); 
// eDataMappingVarNames.battery_SBMU_3_BatteryStatus_ar_CellTemperature_0: 				st_Variable:= IotExtractType(monitor.battery.SBMU[3].BatteryStatus.ar_CellTemperature[0], 1, 0); 
// eDataMappingVarNames.battery_SBMU_0_BatteryStatus_ar_CellTemperature_1: 				st_Variable:= IotExtractType(monitor.battery.SBMU[0].BatteryStatus.ar_CellTemperature[1], 1, 0); 
// eDataMappingVarNames.battery_SBMU_1_BatteryStatus_ar_CellTemperature_1: 				st_Variable:= IotExtractType(monitor.battery.SBMU[1].BatteryStatus.ar_CellTemperature[1], 1, 0); 
// eDataMappingVarNames.battery_SBMU_2_BatteryStatus_ar_CellTemperature_1: 				st_Variable:= IotExtractType(monitor.battery.SBMU[2].BatteryStatus.ar_CellTemperature[1], 1, 0); 
// eDataMappingVarNames.battery_SBMU_3_BatteryStatus_ar_CellTemperature_1: 				st_Variable:= IotExtractType(monitor.battery.SBMU[3].BatteryStatus.ar_CellTemperature[1], 1, 0); 
// eDataMappingVarNames.battery_SBMU_0_BatteryStatus_ar_CellTemperature_2: 				st_Variable:= IotExtractType(monitor.battery.SBMU[0].BatteryStatus.ar_CellTemperature[2], 1, 0); 
// eDataMappingVarNames.battery_SBMU_1_BatteryStatus_ar_CellTemperature_2: 				st_Variable:= IotExtractType(monitor.battery.SBMU[1].BatteryStatus.ar_CellTemperature[2], 1, 0); 
// eDataMappingVarNames.battery_SBMU_2_BatteryStatus_ar_CellTemperature_2: 				st_Variable:= IotExtractType(monitor.battery.SBMU[2].BatteryStatus.ar_CellTemperature[2], 1, 0); 
// eDataMappingVarNames.battery_SBMU_3_BatteryStatus_ar_CellTemperature_2: 				st_Variable:= IotExtractType(monitor.battery.SBMU[3].BatteryStatus.ar_CellTemperature[2], 1, 0); 
// eDataMappingVarNames.battery_SBMU_0_BatteryStatus_r_MaxChargeCurrentAllowed: 				st_Variable:= IotExtractType(monitor.battery.SBMU[0].BatteryStatus.r_MaxChargeCurrentAllowed, 0, 0); 
// eDataMappingVarNames.battery_SBMU_1_BatteryStatus_r_MaxChargeCurrentAllowed: 				st_Variable:= IotExtractType(monitor.battery.SBMU[1].BatteryStatus.r_MaxChargeCurrentAllowed, 0, 0); 
// eDataMappingVarNames.battery_SBMU_2_BatteryStatus_r_MaxChargeCurrentAllowed: 				st_Variable:= IotExtractType(monitor.battery.SBMU[2].BatteryStatus.r_MaxChargeCurrentAllowed, 0, 0); 
// eDataMappingVarNames.battery_SBMU_3_BatteryStatus_r_MaxChargeCurrentAllowed: 				st_Variable:= IotExtractType(monitor.battery.SBMU[3].BatteryStatus.r_MaxChargeCurrentAllowed, 0, 0); 
// eDataMappingVarNames.battery_SBMU_0_BatteryStatus_r_MaxDischargeCurrentAllowed: 				st_Variable:= IotExtractType(monitor.battery.SBMU[0].BatteryStatus.r_MaxDischargeCurrentAllowed, 0, 0); 
// eDataMappingVarNames.battery_SBMU_1_BatteryStatus_r_MaxDischargeCurrentAllowed: 				st_Variable:= IotExtractType(monitor.battery.SBMU[1].BatteryStatus.r_MaxDischargeCurrentAllowed, 0, 0); 
// eDataMappingVarNames.battery_SBMU_2_BatteryStatus_r_MaxDischargeCurrentAllowed: 				st_Variable:= IotExtractType(monitor.battery.SBMU[2].BatteryStatus.r_MaxDischargeCurrentAllowed, 0, 0); 
// eDataMappingVarNames.battery_SBMU_3_BatteryStatus_r_MaxDischargeCurrentAllowed: 				st_Variable:= IotExtractType(monitor.battery.SBMU[3].BatteryStatus.r_MaxDischargeCurrentAllowed, 0, 0); 
// eDataMappingVarNames.battery_SBMU_0_BatteryStatus_r_HistAccChargeEnergy: 				st_Variable:= IotExtractType(monitor.battery.SBMU[0].BatteryStatus.r_HistAccChargeEnergy, 0, 0); 
// eDataMappingVarNames.battery_SBMU_1_BatteryStatus_r_HistAccChargeEnergy: 				st_Variable:= IotExtractType(monitor.battery.SBMU[1].BatteryStatus.r_HistAccChargeEnergy, 0, 0); 
// eDataMappingVarNames.battery_SBMU_2_BatteryStatus_r_HistAccChargeEnergy: 				st_Variable:= IotExtractType(monitor.battery.SBMU[2].BatteryStatus.r_HistAccChargeEnergy, 0, 0); 
// eDataMappingVarNames.battery_SBMU_3_BatteryStatus_r_HistAccChargeEnergy: 				st_Variable:= IotExtractType(monitor.battery.SBMU[3].BatteryStatus.r_HistAccChargeEnergy, 0, 0); 
// eDataMappingVarNames.battery_SBMU_0_BatteryStatus_r_HistAccDischargeEnergy: 				st_Variable:= IotExtractType(monitor.battery.SBMU[0].BatteryStatus.r_HistAccDischargeEnergy, 0, 0); 
// eDataMappingVarNames.battery_SBMU_1_BatteryStatus_r_HistAccDischargeEnergy: 				st_Variable:= IotExtractType(monitor.battery.SBMU[1].BatteryStatus.r_HistAccDischargeEnergy, 0, 0); 
// eDataMappingVarNames.battery_SBMU_2_BatteryStatus_r_HistAccDischargeEnergy: 				st_Variable:= IotExtractType(monitor.battery.SBMU[2].BatteryStatus.r_HistAccDischargeEnergy, 0, 0); 
// eDataMappingVarNames.battery_SBMU_3_BatteryStatus_r_HistAccDischargeEnergy: 				st_Variable:= IotExtractType(monitor.battery.SBMU[3].BatteryStatus.r_HistAccDischargeEnergy, 0, 0); 
// eDataMappingVarNames.battery_SBMU_0_BatteryStatus_w_MaxVoltageCellLocation: 				st_Variable:= IotExtractType(monitor.battery.SBMU[0].BatteryStatus.w_MaxVoltageCellLocation, 0, 0); 
// eDataMappingVarNames.battery_SBMU_1_BatteryStatus_w_MaxVoltageCellLocation: 				st_Variable:= IotExtractType(monitor.battery.SBMU[1].BatteryStatus.w_MaxVoltageCellLocation, 0, 0); 
// eDataMappingVarNames.battery_SBMU_2_BatteryStatus_w_MaxVoltageCellLocation: 				st_Variable:= IotExtractType(monitor.battery.SBMU[2].BatteryStatus.w_MaxVoltageCellLocation, 0, 0); 
// eDataMappingVarNames.battery_SBMU_3_BatteryStatus_w_MaxVoltageCellLocation: 				st_Variable:= IotExtractType(monitor.battery.SBMU[3].BatteryStatus.w_MaxVoltageCellLocation, 0, 0); 
// eDataMappingVarNames.battery_SBMU_0_BatteryStatus_w_MinVoltageCellLocation: 				st_Variable:= IotExtractType(monitor.battery.SBMU[0].BatteryStatus.w_MinVoltageCellLocation, 0, 0); 
// eDataMappingVarNames.battery_SBMU_1_BatteryStatus_w_MinVoltageCellLocation: 				st_Variable:= IotExtractType(monitor.battery.SBMU[1].BatteryStatus.w_MinVoltageCellLocation, 0, 0); 
// eDataMappingVarNames.battery_SBMU_2_BatteryStatus_w_MinVoltageCellLocation: 				st_Variable:= IotExtractType(monitor.battery.SBMU[2].BatteryStatus.w_MinVoltageCellLocation, 0, 0); 
// eDataMappingVarNames.battery_SBMU_3_BatteryStatus_w_MinVoltageCellLocation: 				st_Variable:= IotExtractType(monitor.battery.SBMU[3].BatteryStatus.w_MinVoltageCellLocation, 0, 0); 
// eDataMappingVarNames.battery_SBMU_0_BatteryStatus_w_MaxTempCellLocation: 				st_Variable:= IotExtractType(monitor.battery.SBMU[0].BatteryStatus.w_MaxTempCellLocation, 0, 0); 
// eDataMappingVarNames.battery_SBMU_1_BatteryStatus_w_MaxTempCellLocation: 				st_Variable:= IotExtractType(monitor.battery.SBMU[1].BatteryStatus.w_MaxTempCellLocation, 0, 0); 
// eDataMappingVarNames.battery_SBMU_2_BatteryStatus_w_MaxTempCellLocation: 				st_Variable:= IotExtractType(monitor.battery.SBMU[2].BatteryStatus.w_MaxTempCellLocation, 0, 0); 
// eDataMappingVarNames.battery_SBMU_3_BatteryStatus_w_MaxTempCellLocation: 				st_Variable:= IotExtractType(monitor.battery.SBMU[3].BatteryStatus.w_MaxTempCellLocation, 0, 0); 
// eDataMappingVarNames.battery_SBMU_0_BatteryStatus_w_MinTempCellLocation: 				st_Variable:= IotExtractType(monitor.battery.SBMU[0].BatteryStatus.w_MinTempCellLocation, 0, 0); 
// eDataMappingVarNames.battery_SBMU_1_BatteryStatus_w_MinTempCellLocation: 				st_Variable:= IotExtractType(monitor.battery.SBMU[1].BatteryStatus.w_MinTempCellLocation, 0, 0); 
// eDataMappingVarNames.battery_SBMU_2_BatteryStatus_w_MinTempCellLocation: 				st_Variable:= IotExtractType(monitor.battery.SBMU[2].BatteryStatus.w_MinTempCellLocation, 0, 0); 
// eDataMappingVarNames.battery_SBMU_3_BatteryStatus_w_MinTempCellLocation: 				st_Variable:= IotExtractType(monitor.battery.SBMU[3].BatteryStatus.w_MinTempCellLocation, 0, 0); 
// eDataMappingVarNames.battery_Events_b_COMMUNICATION_ERROR: 				st_Variable:= IotExtractType(monitor.battery.Events.b_COMMUNICATION_ERROR, 0, 0); 
// eDataMappingVarNames.battery_Events_b_OVER_TEMP_ALARM: 				st_Variable:= IotExtractType(monitor.battery.Events.b_OVER_TEMP_ALARM, 0, 0); 
// eDataMappingVarNames.battery_Events_b_OVER_TEMP_WARNING: 				st_Variable:= IotExtractType(monitor.battery.Events.b_OVER_TEMP_WARNING, 0, 0); 
// eDataMappingVarNames.battery_Events_b_UNDER_TEMP_ALARM: 				st_Variable:= IotExtractType(monitor.battery.Events.b_UNDER_TEMP_ALARM, 0, 0); 
// eDataMappingVarNames.battery_Events_b_UNDER_TEMP_WARNING: 				st_Variable:= IotExtractType(monitor.battery.Events.b_UNDER_TEMP_WARNING, 0, 0); 
// eDataMappingVarNames.battery_Events_b_OVER_CHARGE_CURRENT_ALARM: 				st_Variable:= IotExtractType(monitor.battery.Events.b_OVER_CHARGE_CURRENT_ALARM, 0, 0); 
// eDataMappingVarNames.battery_Events_b_OVER_CHARGE_CURRENT_WARNING: 				st_Variable:= IotExtractType(monitor.battery.Events.b_OVER_CHARGE_CURRENT_WARNING, 0, 0); 
// eDataMappingVarNames.battery_Events_b_OVER_DISCHARGE_CURRENT_ALARM: 				st_Variable:= IotExtractType(monitor.battery.Events.b_OVER_DISCHARGE_CURRENT_ALARM, 0, 0); 
// eDataMappingVarNames.battery_Events_b_OVER_DISCHARGE_CURRENT_WARNING: 				st_Variable:= IotExtractType(monitor.battery.Events.b_OVER_DISCHARGE_CURRENT_WARNING, 0, 0); 
// eDataMappingVarNames.battery_Events_b_OVER_VOLT_ALARM: 				st_Variable:= IotExtractType(monitor.battery.Events.b_OVER_VOLT_ALARM, 0, 0); 
// eDataMappingVarNames.battery_Events_b_OVER_VOLT_WARNING: 				st_Variable:= IotExtractType(monitor.battery.Events.b_OVER_VOLT_WARNING, 0, 0); 
// eDataMappingVarNames.battery_Events_b_UNDER_VOLT_ALARM: 				st_Variable:= IotExtractType(monitor.battery.Events.b_UNDER_VOLT_ALARM, 0, 0); 
// eDataMappingVarNames.battery_Events_b_UNDER_VOLT_WARNING: 				st_Variable:= IotExtractType(monitor.battery.Events.b_UNDER_VOLT_WARNING, 0, 0); 
// eDataMappingVarNames.battery_Events_b_UNDER_SOC_MIN_ALARM: 				st_Variable:= IotExtractType(monitor.battery.Events.b_UNDER_SOC_MIN_ALARM, 0, 0); 
// eDataMappingVarNames.battery_Events_b_UNDER_SOC_MIN_WARNING: 				st_Variable:= IotExtractType(monitor.battery.Events.b_UNDER_SOC_MIN_WARNING, 0, 0); 
// eDataMappingVarNames.battery_Events_b_OVER_SOC_MAX_ALARM: 				st_Variable:= IotExtractType(monitor.battery.Events.b_OVER_SOC_MAX_ALARM, 0, 0); 
// eDataMappingVarNames.battery_Events_b_OVER_SOC_MAX_WARNING: 				st_Variable:= IotExtractType(monitor.battery.Events.b_OVER_SOC_MAX_WARNING, 0, 0); 
// eDataMappingVarNames.battery_Events_b_VOLTAGE_IMBALANCE_WARNING: 				st_Variable:= IotExtractType(monitor.battery.Events.b_VOLTAGE_IMBALANCE_WARNING, 0, 0); 
// eDataMappingVarNames.battery_Events_b_TEMPERATURE_IMBALANCE_ALARM: 				st_Variable:= IotExtractType(monitor.battery.Events.b_TEMPERATURE_IMBALANCE_ALARM, 0, 0); 
// eDataMappingVarNames.battery_Events_b_TEMPERATURE_IMBALANCE_WARNING: 				st_Variable:= IotExtractType(monitor.battery.Events.b_TEMPERATURE_IMBALANCE_WARNING, 0, 0); 
// eDataMappingVarNames.battery_Events_b_CONTACTOR_ERROR: 				st_Variable:= IotExtractType(monitor.battery.Events.b_CONTACTOR_ERROR, 0, 0); 
// eDataMappingVarNames.battery_Events_b_FAN_ERROR: 				st_Variable:= IotExtractType(monitor.battery.Events.b_FAN_ERROR, 0, 0); 
// eDataMappingVarNames.battery_Events_b_GROUND_FAULT: 				st_Variable:= IotExtractType(monitor.battery.Events.b_GROUND_FAULT, 0, 0); 
// eDataMappingVarNames.battery_Events_b_OPEN_DOOR_ERROR: 				st_Variable:= IotExtractType(monitor.battery.Events.b_OPEN_DOOR_ERROR, 0, 0); 
// eDataMappingVarNames.battery_Events_b_CURRENT_IMBALANCE_WARNING: 				st_Variable:= IotExtractType(monitor.battery.Events.b_CURRENT_IMBALANCE_WARNING, 0, 0); 
// eDataMappingVarNames.battery_Events_b_OTHER_ALARM: 				st_Variable:= IotExtractType(monitor.battery.Events.b_OTHER_ALARM, 0, 0); 
// eDataMappingVarNames.battery_Events_b_OTHER_WARNING: 				st_Variable:= IotExtractType(monitor.battery.Events.b_OTHER_WARNING, 0, 0); 
// eDataMappingVarNames.battery_Events_b_CONFIGURATION_ALARM: 				st_Variable:= IotExtractType(monitor.battery.Events.b_CONFIGURATION_ALARM, 0, 0); 
// eDataMappingVarNames.battery_Events_b_CONFIGURATION_WARNING: 				st_Variable:= IotExtractType(monitor.battery.Events.b_CONFIGURATION_WARNING, 0, 0); 
// eDataMappingVarNames.battery_Events_b_POWERONFAULT: 				st_Variable:= IotExtractType(monitor.battery.Events.b_POWERONFAULT, 0, 0); 
// eDataMappingVarNames.battery_Events_b_POWEROFFFAULT: 				st_Variable:= IotExtractType(monitor.battery.Events.b_POWEROFFFAULT, 0, 0); 
// eDataMappingVarNames.battery_Events_b_DISCONNECTOR_OFF: 				st_Variable:= IotExtractType(monitor.battery.Events.b_DISCONNECTOR_OFF, 0, 0); 
// eDataMappingVarNames.battery_Events_b_SocLowLimitOutOfRange: 				st_Variable:= IotExtractType(monitor.battery.Events.b_SocLowLimitOutOfRange, 0, 0); 
// eDataMappingVarNames.battery_Events_b_SocHighLimitOutOfRange: 				st_Variable:= IotExtractType(monitor.battery.Events.b_SocHighLimitOutOfRange, 0, 0); 
// eDataMappingVarNames.battery_Events_b_SBMUCommError_0: 				st_Variable:= IotExtractType(monitor.battery.Events.b_SBMUCommError[0], 0, 0); 
// eDataMappingVarNames.battery_Events_b_SBMUCommError_1: 				st_Variable:= IotExtractType(monitor.battery.Events.b_SBMUCommError[1], 0, 0); 
// eDataMappingVarNames.battery_Events_b_SBMUCommError_2: 				st_Variable:= IotExtractType(monitor.battery.Events.b_SBMUCommError[2], 0, 0); 
// eDataMappingVarNames.battery_Events_b_SBMUCommError_3: 				st_Variable:= IotExtractType(monitor.battery.Events.b_SBMUCommError[3], 0, 0); 
// eDataMappingVarNames.battery_Events_b_SBMUFailedToConnect_0: 				st_Variable:= IotExtractType(monitor.battery.Events.b_SBMUFailedToConnect[0], 0, 0); 
// eDataMappingVarNames.battery_Events_b_SBMUFailedToConnect_1: 				st_Variable:= IotExtractType(monitor.battery.Events.b_SBMUFailedToConnect[1], 0, 0); 
// eDataMappingVarNames.battery_Events_b_SBMUFailedToConnect_2: 				st_Variable:= IotExtractType(monitor.battery.Events.b_SBMUFailedToConnect[2], 0, 0); 
// eDataMappingVarNames.battery_Events_b_SBMUFailedToConnect_3: 				st_Variable:= IotExtractType(monitor.battery.Events.b_SBMUFailedToConnect[3], 0, 0); 
// eDataMappingVarNames.protections_FireDetection_b_FireAlarm: 				st_Variable:= IotExtractType(monitor.protections.FireDetection.b_FireAlarm, 0, 0); 
// eDataMappingVarNames.protections_FireDetection_SmokeDetectors_State: 				st_Variable:= IotExtractType(monitor.protections.FireDetection.SmokeDetectors.State, 0, 0); 
// eDataMappingVarNames.protections_FireDetection_CODetectors_State: 				st_Variable:= IotExtractType(monitor.protections.FireDetection.CODetectors.State, 0, 0); 
// eDataMappingVarNames.protections_FireDetection_CODetectors_b_CoValuesOK: 				st_Variable:= IotExtractType(monitor.protections.FireDetection.CODetectors.b_CoValuesOK, 0, 0); 
// eDataMappingVarNames.protections_FireDetection_CODetectors_Value_0: 				st_Variable:= IotExtractType(monitor.protections.FireDetection.CODetectors.Value[0], 1, 0); 
// eDataMappingVarNames.protections_FireDetection_CODetectors_Value_1: 				st_Variable:= IotExtractType(monitor.protections.FireDetection.CODetectors.Value[1], 1, 0); 
// eDataMappingVarNames.protections_FireDetection_CODetectors_Value_2: 				st_Variable:= IotExtractType(monitor.protections.FireDetection.CODetectors.Value[2], 1, 0); 
// eDataMappingVarNames.protections_FireDetection_CODetectors_Value_3: 				st_Variable:= IotExtractType(monitor.protections.FireDetection.CODetectors.Value[3], 1, 0); 
// eDataMappingVarNames.protections_FireDetection_Events_CODetFault: 				st_Variable:= IotExtractType(monitor.protections.FireDetection.Events.CODetFault, 0, 0); 
// eDataMappingVarNames.protections_FireDetection_Events_CODetWarning1: 				st_Variable:= IotExtractType(monitor.protections.FireDetection.Events.CODetWarning1, 0, 0); 
// eDataMappingVarNames.protections_FireDetection_Events_CODetWarning2: 				st_Variable:= IotExtractType(monitor.protections.FireDetection.Events.CODetWarning2, 0, 0); 
// eDataMappingVarNames.protections_FireDetection_Events_CODetAlarm: 				st_Variable:= IotExtractType(monitor.protections.FireDetection.Events.CODetAlarm, 0, 0); 
// eDataMappingVarNames.protections_FireDetection_Events_SmokeDetFault: 				st_Variable:= IotExtractType(monitor.protections.FireDetection.Events.SmokeDetFault, 0, 0); 
// eDataMappingVarNames.protections_FireDetection_Events_SmokeDetAlarm: 				st_Variable:= IotExtractType(monitor.protections.FireDetection.Events.SmokeDetAlarm, 0, 0); 
// eDataMappingVarNames.protections_FireDetection_Events_AlarmMuted: 				st_Variable:= IotExtractType(monitor.protections.FireDetection.Events.AlarmMuted, 0, 0); 
// eDataMappingVarNames.protections_Insulation_b_Enabled: 				st_Variable:= IotExtractType(monitor.protections.Insulation.b_Enabled, 0, 0); 
// eDataMappingVarNames.protections_Insulation_b_PENlinkDetected: 				st_Variable:= IotExtractType(monitor.protections.Insulation.b_PENlinkDetected, 0, 0); 
// eDataMappingVarNames.protections_Insulation_b_Warning: 				st_Variable:= IotExtractType(monitor.protections.Insulation.b_Warning, 0, 0); 
// eDataMappingVarNames.protections_Insulation_e_EarthingSystemDetected: 				st_Variable:= IotExtractType(monitor.protections.Insulation.e_EarthingSystemDetected, 0, 0); 
// eDataMappingVarNames.protections_Insulation_b_PENlinkOperatedFault: 				st_Variable:= IotExtractType(monitor.protections.Insulation.b_PENlinkOperatedFault, 0, 0); 
// eDataMappingVarNames.protections_Insulation_b_EarthingSystemMismatch: 				st_Variable:= IotExtractType(monitor.protections.Insulation.b_EarthingSystemMismatch, 0, 0); 
// eDataMappingVarNames.protections_Insulation_b_NoEarthingSystemSet: 				st_Variable:= IotExtractType(monitor.protections.Insulation.b_NoEarthingSystemSet, 0, 0); 
// eDataMappingVarNames.protections_MRCDB_b_prewarning: 				st_Variable:= IotExtractType(monitor.protections.MRCDB.b_prewarning, 0, 0); 
// eDataMappingVarNames.protections_Surge_b_Type12_OK: 				st_Variable:= IotExtractType(monitor.protections.Surge.b_Type12_OK, 0, 0); 
// eDataMappingVarNames.protections_Surge_b_Type3_OK: 				st_Variable:= IotExtractType(monitor.protections.Surge.b_Type3_OK, 0, 0); 
// eDataMappingVarNames.protections_OvercurrentProtection_r_TotalOutputCurrentLimit: 				st_Variable:= IotExtractType(monitor.protections.OvercurrentProtection.r_TotalOutputCurrentLimit, 0, 0); 
// eDataMappingVarNames.protections_OvercurrentProtection_r_TotalInputCurrentLimit: 				st_Variable:= IotExtractType(monitor.protections.OvercurrentProtection.r_TotalInputCurrentLimit, 0, 0); 
// eDataMappingVarNames.protections_OvercurrentProtection_b_OutputWarning: 				st_Variable:= IotExtractType(monitor.protections.OvercurrentProtection.b_OutputWarning, 0, 0); 
// eDataMappingVarNames.protections_OvercurrentProtection_b_InputWarning: 				st_Variable:= IotExtractType(monitor.protections.OvercurrentProtection.b_InputWarning, 0, 0); 
// eDataMappingVarNames.protections_OvercurrentProtection_b_OutputAlarm: 				st_Variable:= IotExtractType(monitor.protections.OvercurrentProtection.b_OutputAlarm, 0, 0); 
// eDataMappingVarNames.protections_OvercurrentProtection_b_InputAlarm: 				st_Variable:= IotExtractType(monitor.protections.OvercurrentProtection.b_InputAlarm, 0, 0); 
// eDataMappingVarNames.protections_OvercurrentProtection_r_PeakCurrent: 				st_Variable:= IotExtractType(monitor.protections.OvercurrentProtection.r_PeakCurrent, 0, 0); 
// eDataMappingVarNames.protections_OvercurrentProtection_t_PeakCurrentDuration: 				st_Variable:= IotExtractType(monitor.protections.OvercurrentProtection.t_PeakCurrentDuration, 0, 0); 
// eDataMappingVarNames.protections_OvercurrentProtection_s_locationPeak: 				st_Variable:= IotExtractType(monitor.protections.OvercurrentProtection.s_locationPeak, 0, 0); 
// eDataMappingVarNames.peakshavebox_PSBmode: 				st_Variable:= IotExtractType(monitor.peakshavebox.PSBmode, 0, 0); 
// eDataMappingVarNames.peakshavebox_Powermonitor_ar_ApparentPower_AVG: 				st_Variable:= IotExtractType(monitor.peakshavebox.Powermonitor.ar_ApparentPower[0], 1, 1); 
// eDataMappingVarNames.peakshavebox_Powermonitor_ar_ApparentPower_L1: 				st_Variable:= IotExtractType(monitor.peakshavebox.Powermonitor.ar_ApparentPower[1], 1, 1); 
// eDataMappingVarNames.peakshavebox_Powermonitor_ar_ApparentPower_L2: 				st_Variable:= IotExtractType(monitor.peakshavebox.Powermonitor.ar_ApparentPower[2], 1, 1); 
// eDataMappingVarNames.peakshavebox_Powermonitor_ar_ApparentPower_L3: 				st_Variable:= IotExtractType(monitor.peakshavebox.Powermonitor.ar_ApparentPower[3], 1, 1); 
// eDataMappingVarNames.peakshavebox_Powermonitor_ar_ReactivePower_AVG: 				st_Variable:= IotExtractType(monitor.peakshavebox.Powermonitor.ar_ReactivePower[0], 1, 1); 
// eDataMappingVarNames.peakshavebox_Powermonitor_ar_ReactivePower_L1: 				st_Variable:= IotExtractType(monitor.peakshavebox.Powermonitor.ar_ReactivePower[1], 1, 1); 
// eDataMappingVarNames.peakshavebox_Powermonitor_ar_ReactivePower_L2: 				st_Variable:= IotExtractType(monitor.peakshavebox.Powermonitor.ar_ReactivePower[2], 1, 1); 
// eDataMappingVarNames.peakshavebox_Powermonitor_ar_ReactivePower_L3: 				st_Variable:= IotExtractType(monitor.peakshavebox.Powermonitor.ar_ReactivePower[3], 1, 1); 
// eDataMappingVarNames.peakshavebox_Powermonitor_ar_ActivePower_AVG: 				st_Variable:= IotExtractType(monitor.peakshavebox.Powermonitor.ar_ActivePower[0], 1, 1); 
// eDataMappingVarNames.peakshavebox_Powermonitor_ar_ActivePower_L1: 				st_Variable:= IotExtractType(monitor.peakshavebox.Powermonitor.ar_ActivePower[1], 1, 1); 
// eDataMappingVarNames.peakshavebox_Powermonitor_ar_ActivePower_L2: 				st_Variable:= IotExtractType(monitor.peakshavebox.Powermonitor.ar_ActivePower[2], 1, 1); 
// eDataMappingVarNames.peakshavebox_Powermonitor_ar_ActivePower_L3: 				st_Variable:= IotExtractType(monitor.peakshavebox.Powermonitor.ar_ActivePower[3], 1, 1); 
// eDataMappingVarNames.peakshavebox_Powermonitor_r_EnergyConsumed: 				st_Variable:= IotExtractType(monitor.peakshavebox.Powermonitor.r_EnergyConsumed, 0, 0); 
// eDataMappingVarNames.peakshavebox_Powermonitor_r_EnergySupplied: 				st_Variable:= IotExtractType(monitor.peakshavebox.Powermonitor.r_EnergySupplied, 0, 0); 
// eDataMappingVarNames.peakshavebox_Powermonitor_ar_THD_AVG: 				st_Variable:= IotExtractType(monitor.peakshavebox.Powermonitor.ar_THD[0], 1, 0); 
// eDataMappingVarNames.peakshavebox_Powermonitor_ar_THD_L1: 				st_Variable:= IotExtractType(monitor.peakshavebox.Powermonitor.ar_THD[1], 1, 0); 
// eDataMappingVarNames.peakshavebox_Powermonitor_ar_THD_L2: 				st_Variable:= IotExtractType(monitor.peakshavebox.Powermonitor.ar_THD[2], 1, 0); 
// eDataMappingVarNames.peakshavebox_Powermonitor_ar_THD_L3: 				st_Variable:= IotExtractType(monitor.peakshavebox.Powermonitor.ar_THD[3], 1, 0); 
// eDataMappingVarNames.peakshavebox_Powermonitor_ar_PowerFactor_AVG: 				st_Variable:= IotExtractType(monitor.peakshavebox.Powermonitor.ar_PowerFactor[0], 2, 0); 
// eDataMappingVarNames.peakshavebox_Powermonitor_ar_PowerFactor_L1: 				st_Variable:= IotExtractType(monitor.peakshavebox.Powermonitor.ar_PowerFactor[1], 2, 0); 
// eDataMappingVarNames.peakshavebox_Powermonitor_ar_PowerFactor_L2: 				st_Variable:= IotExtractType(monitor.peakshavebox.Powermonitor.ar_PowerFactor[2], 2, 0); 
// eDataMappingVarNames.peakshavebox_Powermonitor_ar_PowerFactor_L3: 				st_Variable:= IotExtractType(monitor.peakshavebox.Powermonitor.ar_PowerFactor[3], 2, 0); 
// eDataMappingVarNames.peakshavebox_Powermonitor_ar_Current_AVG: 				st_Variable:= IotExtractType(monitor.peakshavebox.Powermonitor.ar_Current[0], 1, 1); 
// eDataMappingVarNames.peakshavebox_Powermonitor_ar_Current_L1: 				st_Variable:= IotExtractType(monitor.peakshavebox.Powermonitor.ar_Current[1], 1, 1); 
// eDataMappingVarNames.peakshavebox_Powermonitor_ar_Current_L2: 				st_Variable:= IotExtractType(monitor.peakshavebox.Powermonitor.ar_Current[2], 1, 1); 
// eDataMappingVarNames.peakshavebox_Powermonitor_ar_Current_L3: 				st_Variable:= IotExtractType(monitor.peakshavebox.Powermonitor.ar_Current[3], 1, 1); 
// eDataMappingVarNames.peakshavebox_Powermonitor_ar_Current_N: 				st_Variable:= IotExtractType(monitor.peakshavebox.Powermonitor.ar_Current[4], 1, 1); 
// eDataMappingVarNames.peakshavebox_Powermonitor_r_CurrentUnbalance: 				st_Variable:= IotExtractType(monitor.peakshavebox.Powermonitor.r_CurrentUnbalance, 1, 0); 
// eDataMappingVarNames.peakshavebox_Powermonitor_e_ACrotationStatus: 				st_Variable:= IotExtractType(monitor.peakshavebox.Powermonitor.e_ACrotationStatus, 0, 0); 
// eDataMappingVarNames.peakshavebox_Powermonitor_ar_PhaseVoltage_AVG: 				st_Variable:= IotExtractType(monitor.peakshavebox.Powermonitor.ar_PhaseVoltage[0], 0, 0); 
// eDataMappingVarNames.peakshavebox_Powermonitor_ar_PhaseVoltage_L1: 				st_Variable:= IotExtractType(monitor.peakshavebox.Powermonitor.ar_PhaseVoltage[1], 1, 1); 
// eDataMappingVarNames.peakshavebox_Powermonitor_ar_PhaseVoltage_L2: 				st_Variable:= IotExtractType(monitor.peakshavebox.Powermonitor.ar_PhaseVoltage[2], 1, 1); 
// eDataMappingVarNames.peakshavebox_Powermonitor_ar_PhaseVoltage_L3: 				st_Variable:= IotExtractType(monitor.peakshavebox.Powermonitor.ar_PhaseVoltage[3], 1, 1); 
// eDataMappingVarNames.peakshavebox_Powermonitor_ar_LineVoltage_AVG: 				st_Variable:= IotExtractType(monitor.peakshavebox.Powermonitor.ar_LineVoltage[0], 1, 1); 
// eDataMappingVarNames.peakshavebox_Powermonitor_ar_LineVoltage_L1: 				st_Variable:= IotExtractType(monitor.peakshavebox.Powermonitor.ar_LineVoltage[1], 1, 1); 
// eDataMappingVarNames.peakshavebox_Powermonitor_ar_LineVoltage_L2: 				st_Variable:= IotExtractType(monitor.peakshavebox.Powermonitor.ar_LineVoltage[2], 1, 1); 
// eDataMappingVarNames.peakshavebox_Powermonitor_ar_LineVoltage_L3: 				st_Variable:= IotExtractType(monitor.peakshavebox.Powermonitor.ar_LineVoltage[3], 1, 1); 
// eDataMappingVarNames.peakshavebox_Powermonitor_li_TimeVoltZeroCrossup: 				st_Variable:= IotExtractType(monitor.peakshavebox.Powermonitor.li_TimeVoltZeroCrossup, 0, 0); 
// eDataMappingVarNames.peakshavebox_Powermonitor_ar_Frequency_AVG: 				st_Variable:= IotExtractType(monitor.peakshavebox.Powermonitor.ar_Frequency[0], 2, 1); 
// eDataMappingVarNames.peakshavebox_Powermonitor_ar_Frequency_L1: 				st_Variable:= IotExtractType(monitor.peakshavebox.Powermonitor.ar_Frequency[1], 2, 1); 
// eDataMappingVarNames.peakshavebox_Powermonitor_ar_Frequency_L2: 				st_Variable:= IotExtractType(monitor.peakshavebox.Powermonitor.ar_Frequency[2], 2, 1); 
// eDataMappingVarNames.peakshavebox_Powermonitor_ar_Frequency_L3: 				st_Variable:= IotExtractType(monitor.peakshavebox.Powermonitor.ar_Frequency[3], 2, 1); 
// eDataMappingVarNames.peakshavebox_Powermonitor_r_VoltageUnbalance: 				st_Variable:= IotExtractType(monitor.peakshavebox.Powermonitor.r_VoltageUnbalance, 1, 0); 
// eDataMappingVarNames.peakshavebox_PowerStatus_b_RotaryField: 				st_Variable:= IotExtractType(monitor.peakshavebox.PowerStatus.b_RotaryField, 0, 0); 
// eDataMappingVarNames.peakshavebox_PowerStatus_b_GeneralWarning: 				st_Variable:= IotExtractType(monitor.peakshavebox.PowerStatus.b_GeneralWarning, 0, 0); 
// eDataMappingVarNames.peakshavebox_PowerStatus_b_GeneralFault: 				st_Variable:= IotExtractType(monitor.peakshavebox.PowerStatus.b_GeneralFault, 0, 0); 
// eDataMappingVarNames.peakshavebox_PowerStatus_b_OverVoltage: 				st_Variable:= IotExtractType(monitor.peakshavebox.PowerStatus.b_OverVoltage, 0, 0); 
// eDataMappingVarNames.peakshavebox_PowerStatus_b_UnderVoltage: 				st_Variable:= IotExtractType(monitor.peakshavebox.PowerStatus.b_UnderVoltage, 0, 0); 
// eDataMappingVarNames.peakshavebox_PowerStatus_b_OverCurrent: 				st_Variable:= IotExtractType(monitor.peakshavebox.PowerStatus.b_OverCurrent, 0, 0); 
// eDataMappingVarNames.peakshavebox_PowerStatus_b_Error_Phase_1: 				st_Variable:= IotExtractType(monitor.peakshavebox.PowerStatus.b_Error_Phase[1], 0, 0); 
// eDataMappingVarNames.peakshavebox_PowerStatus_b_Error_Phase_2: 				st_Variable:= IotExtractType(monitor.peakshavebox.PowerStatus.b_Error_Phase[2], 0, 0); 
// eDataMappingVarNames.peakshavebox_PowerStatus_b_Error_Phase_3: 				st_Variable:= IotExtractType(monitor.peakshavebox.PowerStatus.b_Error_Phase[3], 0, 0); 
// eDataMappingVarNames.peakshavebox_r_MaxCTCurrent: 				st_Variable:= IotExtractType(monitor.peakshavebox.r_MaxCTCurrent, 0, 0); 
// eDataMappingVarNames.peakshavebox_b_buscouplerReady: 				st_Variable:= IotExtractType(monitor.peakshavebox.b_buscouplerReady, 0, 0); 
// eDataMappingVarNames.peakshavebox_b_active: 				st_Variable:= IotExtractType(monitor.peakshavebox.b_active, 0, 0); 
// eDataMappingVarNames.peakshavebox_b_dataOK: 				st_Variable:= IotExtractType(monitor.peakshavebox.b_dataOK, 0, 0); 
// eDataMappingVarNames.peakshavebox_b_ContactorFb: 				st_Variable:= IotExtractType(monitor.peakshavebox.b_ContactorFb, 0, 0); 
// eDataMappingVarNames.peakshavebox_b_SyncFb: 				st_Variable:= IotExtractType(monitor.peakshavebox.b_SyncFb, 0, 0); 
// eDataMappingVarNames.peakshavebox_b_SettingsChangePending: 				st_Variable:= IotExtractType(monitor.peakshavebox.b_SettingsChangePending, 0, 0); 
// eDataMappingVarNames.enclosure_climate_r_Humidity: 				st_Variable:= IotExtractType(monitor.enclosure.climate.r_Humidity, 1, 0); 
// eDataMappingVarNames.enclosure_climate_r_Temperature: 				st_Variable:= IotExtractType(monitor.enclosure.climate.r_Temperature, 1, 0); 
// eDataMappingVarNames.enclosure_climate_events_b_HumidityHigh: 				st_Variable:= IotExtractType(monitor.enclosure.climate.events.b_HumidityHigh, 0, 0); 
// eDataMappingVarNames.enclosure_climate_events_b_HumidityTooHigh: 				st_Variable:= IotExtractType(monitor.enclosure.climate.events.b_HumidityTooHigh, 0, 0); 
// eDataMappingVarNames.enclosure_climate_events_b_TemperatureHigh: 				st_Variable:= IotExtractType(monitor.enclosure.climate.events.b_TemperatureHigh, 0, 0); 
// eDataMappingVarNames.enclosure_climate_events_b_TemperatureTooHigh: 				st_Variable:= IotExtractType(monitor.enclosure.climate.events.b_TemperatureTooHigh, 0, 0); 
// eDataMappingVarNames.enclosure_climate_events_b_TemperatureLow: 				st_Variable:= IotExtractType(monitor.enclosure.climate.events.b_TemperatureLow, 0, 0); 
// eDataMappingVarNames.enclosure_climate_events_b_TemperatureTooLow: 				st_Variable:= IotExtractType(monitor.enclosure.climate.events.b_TemperatureTooLow, 0, 0); 
// eDataMappingVarNames.enclosure_climate_events_b_AIOverrange: 				st_Variable:= IotExtractType(monitor.enclosure.climate.events.b_AIOverrange, 0, 0); 
// eDataMappingVarNames.enclosure_climate_events_b_AIUnderrange: 				st_Variable:= IotExtractType(monitor.enclosure.climate.events.b_AIUnderrange, 0, 0); 
// eDataMappingVarNames.enclosure_climate_events_b_AIError: 				st_Variable:= IotExtractType(monitor.enclosure.climate.events.b_AIError, 0, 0); 
// eDataMappingVarNames.enclosure_climate_events_b_DewpointTooHigh: 				st_Variable:= IotExtractType(monitor.enclosure.climate.events.b_DewpointTooHigh, 0, 0); 
// //eDataMappingVarNames.enclosure_doors_b_ClientpanelDoorClosed: 				st_Variable:= IotExtractType(monitor.enclosure.doors.b_ClientpanelDoorClosed, 0, 0); 
// //eDataMappingVarNames.enclosure_doors_b_ControlPanelDoorClosed: 				st_Variable:= IotExtractType(monitor.enclosure.doors.b_ControlPanelDoorClosed, 0, 0); 
// eDataMappingVarNames.enclosure_ledstrip_b_error: 				st_Variable:= IotExtractType(monitor.enclosure.ledstrip.b_error, 0, 0); 
// eDataMappingVarNames.enclosure_ledstrip_BeckhoffLed: 				st_Variable:= IotExtractType(monitor.enclosure.ledstrip.BeckhoffLed, 0, 0); 
// eDataMappingVarNames.internalpsu_b_24VdcAvailable: 				st_Variable:= IotExtractType(monitor.internalpsu.b_24VdcAvailable, 0, 0); 
// eDataMappingVarNames.internalpsu_b_HVDCAvailable: 				st_Variable:= IotExtractType(monitor.internalpsu.b_HVDCAvailable, 0, 0); 
// eDataMappingVarNames.internalpsu_b_400VACAvailable: 				st_Variable:= IotExtractType(monitor.internalpsu.b_400VACAvailable, 0, 0); 
// //eDataMappingVarNames.internalpsu_e_400VSupplySource: 				st_Variable:= IotExtractType(monitor.internalpsu.e_400VSupplySource, 0, 0); 
// eDataMappingVarNames.internalpsu_UPS_r_InputVoltage: 				st_Variable:= IotExtractType(monitor.internalpsu.UPS.r_InputVoltage, 1, 1); 
// eDataMappingVarNames.internalpsu_UPS_r_OutputVoltage: 				st_Variable:= IotExtractType(monitor.internalpsu.UPS.r_OutputVoltage, 1, 1); 
// eDataMappingVarNames.internalpsu_UPS_r_BatteryVoltage: 				st_Variable:= IotExtractType(monitor.internalpsu.UPS.r_BatteryVoltage, 1, 1); 
// eDataMappingVarNames.internalpsu_UPS_r_OutputCurrent: 				st_Variable:= IotExtractType(monitor.internalpsu.UPS.r_OutputCurrent, 2, 0); 
// eDataMappingVarNames.internalpsu_UPS_ui_SOC: 				st_Variable:= IotExtractType(monitor.internalpsu.UPS.ui_SOC, 0, 0); 
// eDataMappingVarNames.internalpsu_UPS_b_ChargerActive: 				st_Variable:= IotExtractType(monitor.internalpsu.UPS.b_ChargerActive, 0, 0); 
// eDataMappingVarNames.internalpsu_UPS_b_SystemOnBattery: 				st_Variable:= IotExtractType(monitor.internalpsu.UPS.b_SystemOnBattery, 0, 0); 
// eDataMappingVarNames.internalpsu_UPS_b_SystemOnDCInput: 				st_Variable:= IotExtractType(monitor.internalpsu.UPS.b_SystemOnDCInput, 0, 0); 
// eDataMappingVarNames.internalpsu_UPS_Events_b_BatteryLowInfo: 				st_Variable:= IotExtractType(monitor.internalpsu.UPS.Events.b_BatteryLowInfo, 0, 0); 
// eDataMappingVarNames.internalpsu_UPS_Events_b_BatteryLowWarning: 				st_Variable:= IotExtractType(monitor.internalpsu.UPS.Events.b_BatteryLowWarning, 0, 0); 
// eDataMappingVarNames.internalpsu_UPS_Events_b_BatteryLowError: 				st_Variable:= IotExtractType(monitor.internalpsu.UPS.Events.b_BatteryLowError, 0, 0); 
// eDataMappingVarNames.internalpsu_UPS_Events_b_NoBatteryError: 				st_Variable:= IotExtractType(monitor.internalpsu.UPS.Events.b_NoBatteryError, 0, 0); 
// eDataMappingVarNames.internalpsu_UPS_Events_b_InputVoltageWarning: 				st_Variable:= IotExtractType(monitor.internalpsu.UPS.Events.b_InputVoltageWarning, 0, 0); 
// eDataMappingVarNames.internalpsu_Events_b_DCPSUFault: 				st_Variable:= IotExtractType(monitor.internalpsu.Events.b_DCPSUFault, 0, 0); 
// eDataMappingVarNames.internalpsu_Events_b_ACPSUFault: 				st_Variable:= IotExtractType(monitor.internalpsu.Events.b_ACPSUFault, 0, 0); 
// eDataMappingVarNames.internalpsu_Events_b_GridInputFuseTripped: 				st_Variable:= IotExtractType(monitor.internalpsu.Events.b_GridInputFuseTripped, 0, 0); 
// //eDataMappingVarNames.internalpsu_Events_b_CEEInputFuseTripped: 				st_Variable:= IotExtractType(monitor.internalpsu.Events.b_CEEInputFuseTripped, 0, 0); 
// eDataMappingVarNames.internalpsu_Events_b_HVDCShutdownTimeExceeded: 				st_Variable:= IotExtractType(monitor.internalpsu.Events.b_HVDCShutdownTimeExceeded, 0, 0); 
// eDataMappingVarNames.internalpsu_Events_b_UPSLowShutdown: 				st_Variable:= IotExtractType(monitor.internalpsu.Events.b_UPSLowShutdown, 0, 0); 
// eDataMappingVarNames.PLC_r_CPUload: 				st_Variable:= IotExtractType(monitor.PLC.r_CPUload, 0, 0); 
// eDataMappingVarNames.PLC_e_ProfinetState: 				st_Variable:= IotExtractType(monitor.PLC.e_ProfinetState, 0, 0); 
// eDataMappingVarNames.PLC_e_EthercatState: 				st_Variable:= IotExtractType(monitor.PLC.e_EthercatState, 0, 0); 
// eDataMappingVarNames.Cooling_CoolingSystemMode: 				st_Variable:= IotExtractType(monitor.Cooling.CoolingSystemMode, 0, 0); 
// eDataMappingVarNames.Cooling_HeatPumpStatus: 				st_Variable:= IotExtractType(monitor.Cooling.HeatPumpStatus, 0, 0); 
// eDataMappingVarNames.Cooling_r_CoolantTemperature: 				st_Variable:= IotExtractType(monitor.Cooling.r_CoolantTemperature, 1, 0); 
// eDataMappingVarNames.Cooling_r_CoolantPressure: 				st_Variable:= IotExtractType(monitor.Cooling.r_CoolantPressure, 2, 0); 
// eDataMappingVarNames.Cooling_r_EnclosureDewpoint: 				st_Variable:= IotExtractType(monitor.Cooling.r_EnclosureDewpoint, 0, 0); 
// eDataMappingVarNames.Cooling_ui_DehumRemainingTime: 				st_Variable:= IotExtractType(monitor.Cooling.ui_DehumRemainingTime, 0, 0); 
// eDataMappingVarNames.Cooling_HeatPumpSystem_HeatPumpStatus: 				st_Variable:= IotExtractType(monitor.Cooling.HeatPumpStatus, 0, 0); 
// eDataMappingVarNames.Cooling_HeatPumpSystem_PrimaryHeatpumpGet_HeatPumpState: 				st_Variable:= IotExtractType(monitor.Cooling.HeatPumpStatus, 0, 0); {warning 'needs revision, heatpump now doesn't have individuals state'} 
// eDataMappingVarNames.Cooling_HeatPumpSystem_PrimaryHeatpumpGet_Setpoint: 				st_Variable:= IotExtractType(monitor.Cooling.Heatpump.Setpoint, 0, 0); 
// eDataMappingVarNames.Cooling_HeatPumpSystem_PrimaryHeatpumpGet_Events_b_CommWarning: 				st_Variable:= IotExtractType(monitor.Cooling.Heatpump.Events.b_CommWarning, 0, 0); 
// eDataMappingVarNames.Cooling_HeatPumpSystem_PrimaryHeatpumpGet_Events_b_ProbeError: 				st_Variable:= IotExtractType(monitor.Cooling.Heatpump.Events.b_ProbeError, 0, 0); 
// eDataMappingVarNames.Cooling_HeatPumpSystem_PrimaryHeatpumpGet_Events_b_PressureError: 				st_Variable:= IotExtractType(monitor.Cooling.Heatpump.Events.b_PressureError, 0, 0); 
// eDataMappingVarNames.Cooling_HeatPumpSystem_PrimaryHeatpumpGet_Events_b_CompressorError: 				st_Variable:= IotExtractType(monitor.Cooling.Heatpump.Events.b_CompressorError, 0, 0); 
// eDataMappingVarNames.Cooling_HeatPumpSystem_PrimaryHeatpumpGet_Events_b_ValveError: 				st_Variable:= IotExtractType(monitor.Cooling.Heatpump.Events.b_ValveError, 0, 0); 
// eDataMappingVarNames.Cooling_HeatPumpSystem_PrimaryHeatpumpGet_Events_b_FanError: 				st_Variable:= IotExtractType(monitor.Cooling.Heatpump.Events.b_FanError, 0, 0); 
// eDataMappingVarNames.Cooling_HeatPumpSystem_PrimaryHeatpumpGet_Events_b_PumpError: 				st_Variable:= IotExtractType(monitor.Cooling.Heatpump.Events.b_PumpError, 0, 0); 
// eDataMappingVarNames.Cooling_HeatPumpSystem_PrimaryHeatpumpGet_Events_b_WaterTempError: 				st_Variable:= IotExtractType(monitor.Cooling.Heatpump.Events.b_WaterTempError, 0, 0); 
// eDataMappingVarNames.Cooling_HeatPumpSystem_PrimaryHeatpumpGet_Events_b_IOError: 				st_Variable:= IotExtractType(monitor.Cooling.Heatpump.Events.b_IOError, 0, 0); 
// eDataMappingVarNames.Cooling_HeatPumpSystem_PrimaryHeatpumpGet_Events_b_HeatpumpPreheatingActive: 				st_Variable:= IotExtractType(monitor.Cooling.Heatpump.Events.b_HeatpumpPreheatingActive, 0, 0); 
// eDataMappingVarNames.Cooling_HeatPumpSystem_PrimaryHeatpumpGet_Events_b_TooColdForHeatpumpHeating: 				st_Variable:= IotExtractType(monitor.Cooling.Heatpump.Events.b_TooColdForHeatpumpHeating, 0, 0); 
// eDataMappingVarNames.Cooling_HeatPumpSystem_PrimaryHeatpumpGet_HeatpumpData_i_FW_Version: 				st_Variable:= IotExtractType(monitor.Cooling.Heatpump.HeatpumpData.i_FW_Version, 0, 0); 
// eDataMappingVarNames.Cooling_HeatPumpSystem_PrimaryHeatpumpGet_HeatpumpData_i_FW_release: 				st_Variable:= IotExtractType(monitor.Cooling.Heatpump.HeatpumpData.i_FW_release, 0, 0); 
// eDataMappingVarNames.Cooling_HeatPumpSystem_PrimaryHeatpumpGet_HeatpumpData_w_FW_Subrelease: 				st_Variable:= IotExtractType(monitor.Cooling.Heatpump.HeatpumpData.HeatpumpData.w_FW_Subrelease, 0, 0); 
// eDataMappingVarNames.Cooling_HeatPumpSystem_PrimaryHeatpumpGet_HeatpumpData_w_FW_creationDate: 				st_Variable:= IotExtractType(monitor.Cooling.Heatpump.Heatpumpdata.w_FW_creationDate, 0, 0); 
// eDataMappingVarNames.Cooling_HeatPumpSystem_PrimaryHeatpumpGet_HeatpumpData_w_Serialnumber_0: 				st_Variable:= IotExtractType(monitor.Cooling.Heatpump.Heatpumpdata.w_Serialnumber[0], 0, 0); 
// eDataMappingVarNames.Cooling_HeatPumpSystem_PrimaryHeatpumpGet_HeatpumpData_w_Serialnumber_1: 				st_Variable:= IotExtractType(monitor.Cooling.Heatpump.Heatpumpdata.w_Serialnumber[1], 0, 0); 
// eDataMappingVarNames.Cooling_HeatPumpSystem_PrimaryHeatpumpGet_HeatpumpData_w_Serialnumber_2: 				st_Variable:= IotExtractType(monitor.Cooling.Heatpump.Heatpumpdata.w_Serialnumber[2], 0, 0); 
// eDataMappingVarNames.Cooling_HeatPumpSystem_PrimaryHeatpumpGet_HeatpumpData_w_Serialnumber_3: 				st_Variable:= IotExtractType(monitor.Cooling.Heatpump.Heatpumpdata.w_Serialnumber[3], 0, 0); 
// eDataMappingVarNames.Cooling_HeatPumpSystem_PrimaryHeatpumpGet_HeatpumpData_w_Serialnumber_4: 				st_Variable:= IotExtractType(monitor.Cooling.Heatpump.Heatpumpdata.w_Serialnumber[4], 0, 0); 
// eDataMappingVarNames.Cooling_HeatPumpSystem_PrimaryHeatpumpGet_HeatpumpData_w_Serialnumber_5: 				st_Variable:= IotExtractType(monitor.Cooling.Heatpump.Heatpumpdata.w_Serialnumber[5], 0, 0); 
// eDataMappingVarNames.Cooling_HeatPumpSystem_PrimaryHeatpumpGet_HeatpumpData_w_Serialnumber_6: 				st_Variable:= IotExtractType(monitor.Cooling.Heatpump.Heatpumpdata.w_Serialnumber[6], 0, 0); 
// eDataMappingVarNames.Cooling_HeatPumpSystem_PrimaryHeatpumpGet_HeatpumpData_w_Serialnumber_7: 				st_Variable:= IotExtractType(monitor.Cooling.Heatpump.Heatpumpdata.w_Serialnumber[7], 0, 0); 
// eDataMappingVarNames.Cooling_HeatPumpSystem_PrimaryHeatpumpGet_HeatpumpData_w_Serialnumber_8: 				st_Variable:= IotExtractType(monitor.Cooling.Heatpump.Heatpumpdata.w_Serialnumber[8], 0, 0); 
// eDataMappingVarNames.Cooling_HeatPumpSystem_PrimaryHeatpumpGet_HeatpumpData_w_Serialnumber_9: 				st_Variable:= IotExtractType(monitor.Cooling.Heatpump.Heatpumpdata.w_Serialnumber[9], 0, 0); 
// eDataMappingVarNames.Cooling_HeatPumpSystem_PrimaryHeatpumpGet_HeatpumpData_w_Serialnumber_10: 				st_Variable:= IotExtractType(monitor.Cooling.Heatpump.Heatpumpdata.w_Serialnumber[10], 0, 0); 
// eDataMappingVarNames.Cooling_HeatPumpSystem_PrimaryHeatpumpGet_HeatpumpData_w_Serialnumber_11: 				st_Variable:= IotExtractType(monitor.Cooling.Heatpump.Heatpumpdata.w_Serialnumber[11], 0, 0); 
// eDataMappingVarNames.Cooling_HeatPumpSystem_PrimaryHeatpumpGet_HeatpumpData_w_Serialnumber_12: 				st_Variable:= IotExtractType(monitor.Cooling.Heatpump.Heatpumpdata.w_Serialnumber[12], 0, 0); 
// eDataMappingVarNames.Cooling_HeatPumpSystem_PrimaryHeatpumpGet_HeatpumpData_w_Serialnumber_13: 				st_Variable:= IotExtractType(monitor.Cooling.Heatpump.Heatpumpdata.w_Serialnumber[13], 0, 0); 
// eDataMappingVarNames.Cooling_HeatPumpSystem_PrimaryHeatpumpGet_HeatpumpData_w_Serialnumber_14: 				st_Variable:= IotExtractType(monitor.Cooling.Heatpump.Heatpumpdata.w_Serialnumber[14], 0, 0); 
// eDataMappingVarNames.Cooling_HeatPumpSystem_PrimaryHeatpumpGet_HeatpumpData_w_Serialnumber_15: 				st_Variable:= IotExtractType(monitor.Cooling.Heatpump.Heatpumpdata.w_Serialnumber[15], 0, 0); 
// eDataMappingVarNames.Cooling_HeatPumpSystem_PrimaryHeatpumpGet_HeatpumpData_w_Serialnumber_16: 				st_Variable:= IotExtractType(monitor.Cooling.Heatpump.Heatpumpdata.w_Serialnumber[16], 0, 0); 
// eDataMappingVarNames.Cooling_HeatPumpSystem_PrimaryHeatpumpGet_HeatpumpData_w_Serialnumber_17: 				st_Variable:= IotExtractType(monitor.Cooling.Heatpump.Heatpumpdata.w_Serialnumber[17], 0, 0); 
// eDataMappingVarNames.Cooling_HeatPumpSystem_PrimaryHeatpumpGet_HeatpumpData_i_OperatingHours: 				st_Variable:= IotExtractType(monitor.Cooling.Heatpump.Heatpumpdata.i_OperatingHours, 0, 0); 
// eDataMappingVarNames.Cooling_HeatPumpSystem_PrimaryHeatpumpGet_HeatpumpData_r_CoolantPower: 				st_Variable:= IotExtractType(monitor.Cooling.Heatpump.Heatpumpdata.r_CoolantPower, 0, 0); 
// eDataMappingVarNames.Cooling_HeatPumpSystem_PrimaryHeatpumpGet_HeatpumpData_r_InletWaterTemp: 				st_Variable:= IotExtractType(monitor.Cooling.Heatpump.Heatpumpdata.r_InletWaterTemp, 0, 0); 
// eDataMappingVarNames.Cooling_HeatPumpSystem_PrimaryHeatpumpGet_HeatpumpData_r_OutletWaterTemp: 				st_Variable:= IotExtractType(monitor.Cooling.Heatpump.Heatpumpdata.r_OutletWaterTemp, 0, 0); 
// eDataMappingVarNames.Cooling_HeatPumpSystem_PrimaryHeatpumpGet_HeatpumpData_r_HighPressure: 				st_Variable:= IotExtractType(monitor.Cooling.Heatpump.Heatpumpdata.r_HighPressure, 0, 0); 
// eDataMappingVarNames.Cooling_HeatPumpSystem_PrimaryHeatpumpGet_HeatpumpData_r_LowPressure: 				st_Variable:= IotExtractType(monitor.Cooling.HeatPump.HeatpumpData.r_LowPressure, 0, 0); 
// eDataMappingVarNames.Cooling_HeatPumpSystem_PrimaryHeatpumpGet_HeatpumpData_r_CompInputTemp: 				st_Variable:= IotExtractType(monitor.Cooling.Heatpump.HeatpumpData.r_CompInputTemp, 0, 0); 
// eDataMappingVarNames.Cooling_HeatPumpSystem_PrimaryHeatpumpGet_HeatpumpData_r_OutdoorTemp: 				st_Variable:= IotExtractType(monitor.Cooling.Heatpump.HeatpumpData.r_OutdoorTemp, 0, 0); 
// eDataMappingVarNames.Cooling_HeatPumpSystem_PrimaryHeatpumpGet_HeatpumpData_r_CompOutputTemp: 				st_Variable:= IotExtractType(monitor.Cooling.Heatpump.HeatpumpData.r_CompOutputTemp, 0, 0); 
// eDataMappingVarNames.Cooling_HeatPumpSystem_PrimaryHeatpumpGet_HeatpumpData_ui_WaterFlowRate: 				st_Variable:= IotExtractType(monitor.Cooling.Heatpump.HeatpumpData.ui_WaterFlowRate, 0, 0); 
// eDataMappingVarNames.Cooling_HeatPumpSystem_PrimaryHeatpumpGet_HeatpumpData_w_ErrorList_1: 				st_Variable:= IotExtractType(monitor.Cooling.Heatpump.HeatpumpData.w_ErrorList[1], 0, 0); 
// eDataMappingVarNames.Cooling_HeatPumpSystem_PrimaryHeatpumpGet_HeatpumpData_w_ErrorList_2: 				st_Variable:= IotExtractType(monitor.Cooling.Heatpump.HeatpumpData.w_ErrorList[2], 0, 0); 
// eDataMappingVarNames.Cooling_HeatPumpSystem_PrimaryHeatpumpGet_HeatpumpData_w_ErrorList_3: 				st_Variable:= IotExtractType(monitor.Cooling.Heatpump.HeatpumpData.w_ErrorList[3], 0, 0); 
// eDataMappingVarNames.Cooling_HeatPumpSystem_PrimaryHeatpumpGet_HeatpumpData_w_ErrorList_4: 				st_Variable:= IotExtractType(monitor.Cooling.Heatpump.HeatpumpData.w_ErrorList[4], 0, 0); 
// eDataMappingVarNames.Cooling_HeatPumpSystem_PrimaryHeatpumpGet_HeatpumpData_w_ErrorList_5: 				st_Variable:= IotExtractType(monitor.Cooling.Heatpump.HeatpumpData.w_ErrorList[5], 0, 0); 
// eDataMappingVarNames.Cooling_HeatPumpSystem_PrimaryHeatpumpGet_HeatpumpData_w_ErrorList_6: 				st_Variable:= IotExtractType(monitor.Cooling.Heatpump.HeatpumpData.w_ErrorList[6], 0, 0); 
// eDataMappingVarNames.Cooling_HeatPumpSystem_PrimaryHeatpumpGet_HeatpumpData_w_ErrorList_7: 				st_Variable:= IotExtractType(monitor.Cooling.Heatpump.HeatpumpData.w_ErrorList[7], 0, 0); 
// eDataMappingVarNames.Cooling_HeatPumpSystem_PrimaryHeatpumpGet_HeatpumpData_r_FanSpeedPCT: 				st_Variable:= IotExtractType(monitor.Cooling.Heatpump.HeatpumpData.r_FanSpeedPCT, 0, 0); 
// eDataMappingVarNames.Cooling_HeatPumpSystem_PrimaryHeatpumpGet_HeatpumpData_r_PumpSpeedPCT: 				st_Variable:= IotExtractType(monitor.Cooling.Heatpump.HeatpumpData.r_PumpSpeedPCT, 0, 0); 
// eDataMappingVarNames.Cooling_HeatPumpSystem_PrimaryHeatpumpGet_HeatpumpData_r_SetpointHeating: 				st_Variable:= IotExtractType(monitor.Cooling.Heatpump.HeatpumpData.r_SetpointHeating, 1, 0); 
// eDataMappingVarNames.Cooling_HeatPumpSystem_PrimaryHeatpumpGet_HeatpumpData_r_SetpointCooling: 				st_Variable:= IotExtractType(monitor.Cooling.Heatpump.HeatpumpData.r_SetpointCooling, 1, 0); 
// eDataMappingVarNames.Cooling_HeatPumpSystem_PrimaryHeatpumpGet_HeatpumpData_b_DefrostingActive: 				st_Variable:= IotExtractType(monitor.Cooling.Heatpump.HeatpumpData.b_DefrostingActive, 0, 0); 
// eDataMappingVarNames.Cooling_HeatPumpSystem_SecondaryHeatpumpGet_HeatPumpState: 				st_Variable:= IotExtractType(monitor.Cooling.HeatPumpSystem.SecondaryHeatpumpGet.HeatPumpState, 0, 0); 
// eDataMappingVarNames.Cooling_HeatPumpSystem_SecondaryHeatpumpGet_Setpoint: 				st_Variable:= IotExtractType(monitor.Cooling.HeatPumpSystem.SecondaryHeatpumpGet.Setpoint, 0, 0); 
// eDataMappingVarNames.Cooling_HeatPumpSystem_SecondaryHeatpumpGet_Events_b_CommWarning: 				st_Variable:= IotExtractType(monitor.Cooling.HeatPumpSystem.SecondaryHeatpumpGet.Events.b_CommWarning, 0, 0); 
// eDataMappingVarNames.Cooling_HeatPumpSystem_SecondaryHeatpumpGet_Events_b_ProbeError: 				st_Variable:= IotExtractType(monitor.Cooling.HeatPumpSystem.SecondaryHeatpumpGet.Events.b_ProbeError, 0, 0); 
// eDataMappingVarNames.Cooling_HeatPumpSystem_SecondaryHeatpumpGet_Events_b_PressureError: 				st_Variable:= IotExtractType(monitor.Cooling.HeatPumpSystem.SecondaryHeatpumpGet.Events.b_PressureError, 0, 0); 
// eDataMappingVarNames.Cooling_HeatPumpSystem_SecondaryHeatpumpGet_Events_b_CompressorError: 				st_Variable:= IotExtractType(monitor.Cooling.HeatPumpSystem.SecondaryHeatpumpGet.Events.b_CompressorError, 0, 0); 
// eDataMappingVarNames.Cooling_HeatPumpSystem_SecondaryHeatpumpGet_Events_b_ValveError: 				st_Variable:= IotExtractType(monitor.Cooling.HeatPumpSystem.SecondaryHeatpumpGet.Events.b_ValveError, 0, 0); 
// eDataMappingVarNames.Cooling_HeatPumpSystem_SecondaryHeatpumpGet_Events_b_FanError: 				st_Variable:= IotExtractType(monitor.Cooling.HeatPumpSystem.SecondaryHeatpumpGet.Events.b_FanError, 0, 0); 
// eDataMappingVarNames.Cooling_HeatPumpSystem_SecondaryHeatpumpGet_Events_b_PumpError: 				st_Variable:= IotExtractType(monitor.Cooling.HeatPumpSystem.SecondaryHeatpumpGet.Events.b_PumpError, 0, 0); 
// eDataMappingVarNames.Cooling_HeatPumpSystem_SecondaryHeatpumpGet_Events_b_WaterTempError: 				st_Variable:= IotExtractType(monitor.Cooling.HeatPumpSystem.SecondaryHeatpumpGet.Events.b_WaterTempError, 0, 0); 
// eDataMappingVarNames.Cooling_HeatPumpSystem_SecondaryHeatpumpGet_Events_b_IOError: 				st_Variable:= IotExtractType(monitor.Cooling.HeatPumpSystem.SecondaryHeatpumpGet.Events.b_IOError, 0, 0); 
// eDataMappingVarNames.Cooling_HeatPumpSystem_SecondaryHeatpumpGet_Events_b_HeatpumpPreheatingActive: 				st_Variable:= IotExtractType(monitor.Cooling.HeatPumpSystem.SecondaryHeatpumpGet.Events.b_HeatpumpPreheatingActive, 0, 0); 
// eDataMappingVarNames.Cooling_HeatPumpSystem_SecondaryHeatpumpGet_Events_b_TooColdForHeatpumpHeating: 				st_Variable:= IotExtractType(monitor.Cooling.HeatPumpSystem.SecondaryHeatpumpGet.Events.b_TooColdForHeatpumpHeating, 0, 0); 
// eDataMappingVarNames.Cooling_HeatPumpSystem_SecondaryHeatpumpGet_HeatpumpData_i_FW_Version: 				st_Variable:= IotExtractType(monitor.Cooling.HeatPumpSystem.SecondaryHeatpumpGet.HeatpumpData.i_FW_Version, 0, 0); 
// eDataMappingVarNames.Cooling_HeatPumpSystem_SecondaryHeatpumpGet_HeatpumpData_i_FW_release: 				st_Variable:= IotExtractType(monitor.Cooling.HeatPumpSystem.SecondaryHeatpumpGet.HeatpumpData.i_FW_release, 0, 0); 
// eDataMappingVarNames.Cooling_HeatPumpSystem_SecondaryHeatpumpGet_HeatpumpData_w_FW_Subrelease: 				st_Variable:= IotExtractType(monitor.Cooling.HeatPumpSystem.SecondaryHeatpumpGet.HeatpumpData.w_FW_Subrelease, 0, 0); 
// eDataMappingVarNames.Cooling_HeatPumpSystem_SecondaryHeatpumpGet_HeatpumpData_w_FW_creationDate: 				st_Variable:= IotExtractType(monitor.Cooling.HeatPumpSystem.SecondaryHeatpumpGet.HeatpumpData.w_FW_creationDate, 0, 0); 
// eDataMappingVarNames.Cooling_HeatPumpSystem_SecondaryHeatpumpGet_HeatpumpData_w_Serialnumber_0: 				st_Variable:= IotExtractType(monitor.Cooling.HeatPumpSystem.SecondaryHeatpumpGet.HeatpumpData.w_Serialnumber[0], 0, 0); 
// eDataMappingVarNames.Cooling_HeatPumpSystem_SecondaryHeatpumpGet_HeatpumpData_w_Serialnumber_1: 				st_Variable:= IotExtractType(monitor.Cooling.HeatPumpSystem.SecondaryHeatpumpGet.HeatpumpData.w_Serialnumber[1], 0, 0); 
// eDataMappingVarNames.Cooling_HeatPumpSystem_SecondaryHeatpumpGet_HeatpumpData_w_Serialnumber_2: 				st_Variable:= IotExtractType(monitor.Cooling.HeatPumpSystem.SecondaryHeatpumpGet.HeatpumpData.w_Serialnumber[2], 0, 0); 
// eDataMappingVarNames.Cooling_HeatPumpSystem_SecondaryHeatpumpGet_HeatpumpData_w_Serialnumber_3: 				st_Variable:= IotExtractType(monitor.Cooling.HeatPumpSystem.SecondaryHeatpumpGet.HeatpumpData.w_Serialnumber[3], 0, 0); 
// eDataMappingVarNames.Cooling_HeatPumpSystem_SecondaryHeatpumpGet_HeatpumpData_w_Serialnumber_4: 				st_Variable:= IotExtractType(monitor.Cooling.HeatPumpSystem.SecondaryHeatpumpGet.HeatpumpData.w_Serialnumber[4], 0, 0); 
// eDataMappingVarNames.Cooling_HeatPumpSystem_SecondaryHeatpumpGet_HeatpumpData_w_Serialnumber_5: 				st_Variable:= IotExtractType(monitor.Cooling.HeatPumpSystem.SecondaryHeatpumpGet.HeatpumpData.w_Serialnumber[5], 0, 0); 
// eDataMappingVarNames.Cooling_HeatPumpSystem_SecondaryHeatpumpGet_HeatpumpData_w_Serialnumber_6: 				st_Variable:= IotExtractType(monitor.Cooling.HeatPumpSystem.SecondaryHeatpumpGet.HeatpumpData.w_Serialnumber[6], 0, 0); 
// eDataMappingVarNames.Cooling_HeatPumpSystem_SecondaryHeatpumpGet_HeatpumpData_w_Serialnumber_7: 				st_Variable:= IotExtractType(monitor.Cooling.HeatPumpSystem.SecondaryHeatpumpGet.HeatpumpData.w_Serialnumber[7], 0, 0); 
// eDataMappingVarNames.Cooling_HeatPumpSystem_SecondaryHeatpumpGet_HeatpumpData_w_Serialnumber_8: 				st_Variable:= IotExtractType(monitor.Cooling.HeatPumpSystem.SecondaryHeatpumpGet.HeatpumpData.w_Serialnumber[8], 0, 0); 
// eDataMappingVarNames.Cooling_HeatPumpSystem_SecondaryHeatpumpGet_HeatpumpData_w_Serialnumber_9: 				st_Variable:= IotExtractType(monitor.Cooling.HeatPumpSystem.SecondaryHeatpumpGet.HeatpumpData.w_Serialnumber[9], 0, 0); 
// eDataMappingVarNames.Cooling_HeatPumpSystem_SecondaryHeatpumpGet_HeatpumpData_w_Serialnumber_10: 				st_Variable:= IotExtractType(monitor.Cooling.HeatPumpSystem.SecondaryHeatpumpGet.HeatpumpData.w_Serialnumber[10], 0, 0); 
// eDataMappingVarNames.Cooling_HeatPumpSystem_SecondaryHeatpumpGet_HeatpumpData_w_Serialnumber_11: 				st_Variable:= IotExtractType(monitor.Cooling.HeatPumpSystem.SecondaryHeatpumpGet.HeatpumpData.w_Serialnumber[11], 0, 0); 
// eDataMappingVarNames.Cooling_HeatPumpSystem_SecondaryHeatpumpGet_HeatpumpData_w_Serialnumber_12: 				st_Variable:= IotExtractType(monitor.Cooling.HeatPumpSystem.SecondaryHeatpumpGet.HeatpumpData.w_Serialnumber[12], 0, 0); 
// eDataMappingVarNames.Cooling_HeatPumpSystem_SecondaryHeatpumpGet_HeatpumpData_w_Serialnumber_13: 				st_Variable:= IotExtractType(monitor.Cooling.HeatPumpSystem.SecondaryHeatpumpGet.HeatpumpData.w_Serialnumber[13], 0, 0); 
// eDataMappingVarNames.Cooling_HeatPumpSystem_SecondaryHeatpumpGet_HeatpumpData_w_Serialnumber_14: 				st_Variable:= IotExtractType(monitor.Cooling.HeatPumpSystem.SecondaryHeatpumpGet.HeatpumpData.w_Serialnumber[14], 0, 0); 
// eDataMappingVarNames.Cooling_HeatPumpSystem_SecondaryHeatpumpGet_HeatpumpData_w_Serialnumber_15: 				st_Variable:= IotExtractType(monitor.Cooling.HeatPumpSystem.SecondaryHeatpumpGet.HeatpumpData.w_Serialnumber[15], 0, 0); 
// eDataMappingVarNames.Cooling_HeatPumpSystem_SecondaryHeatpumpGet_HeatpumpData_w_Serialnumber_16: 				st_Variable:= IotExtractType(monitor.Cooling.HeatPumpSystem.SecondaryHeatpumpGet.HeatpumpData.w_Serialnumber[16], 0, 0); 
// eDataMappingVarNames.Cooling_HeatPumpSystem_SecondaryHeatpumpGet_HeatpumpData_w_Serialnumber_17: 				st_Variable:= IotExtractType(monitor.Cooling.HeatPumpSystem.SecondaryHeatpumpGet.HeatpumpData.w_Serialnumber[17], 0, 0); 
// eDataMappingVarNames.Cooling_HeatPumpSystem_SecondaryHeatpumpGet_HeatpumpData_i_OperatingHours: 				st_Variable:= IotExtractType(monitor.Cooling.HeatPumpSystem.SecondaryHeatpumpGet.HeatpumpData.i_OperatingHours, 0, 0); 
// eDataMappingVarNames.Cooling_HeatPumpSystem_SecondaryHeatpumpGet_HeatpumpData_r_CoolantPower: 				st_Variable:= IotExtractType(monitor.Cooling.HeatPumpSystem.SecondaryHeatpumpGet.HeatpumpData.r_CoolantPower, 1, 0); 
// eDataMappingVarNames.Cooling_HeatPumpSystem_SecondaryHeatpumpGet_HeatpumpData_r_InletWaterTemp: 				st_Variable:= IotExtractType(monitor.Cooling.HeatPumpSystem.SecondaryHeatpumpGet.HeatpumpData.r_InletWaterTemp, 1, 0); 
// eDataMappingVarNames.Cooling_HeatPumpSystem_SecondaryHeatpumpGet_HeatpumpData_r_OutletWaterTemp: 				st_Variable:= IotExtractType(monitor.Cooling.HeatPumpSystem.SecondaryHeatpumpGet.HeatpumpData.r_OutletWaterTemp, 1, 0); 
// eDataMappingVarNames.Cooling_HeatPumpSystem_SecondaryHeatpumpGet_HeatpumpData_r_HighPressure: 				st_Variable:= IotExtractType(monitor.Cooling.HeatPumpSystem.SecondaryHeatpumpGet.HeatpumpData.r_HighPressure, 1, 0); 
// eDataMappingVarNames.Cooling_HeatPumpSystem_SecondaryHeatpumpGet_HeatpumpData_r_LowPressure: 				st_Variable:= IotExtractType(monitor.Cooling.HeatPumpSystem.SecondaryHeatpumpGet.HeatpumpData.r_LowPressure, 1, 0); 
// eDataMappingVarNames.Cooling_HeatPumpSystem_SecondaryHeatpumpGet_HeatpumpData_r_CompInputTemp: 				st_Variable:= IotExtractType(monitor.Cooling.HeatPumpSystem.SecondaryHeatpumpGet.HeatpumpData.r_CompInputTemp, 1, 0); 
// eDataMappingVarNames.Cooling_HeatPumpSystem_SecondaryHeatpumpGet_HeatpumpData_r_OutdoorTemp: 				st_Variable:= IotExtractType(monitor.Cooling.HeatPumpSystem.SecondaryHeatpumpGet.HeatpumpData.r_OutdoorTemp, 1, 0); 
// eDataMappingVarNames.Cooling_HeatPumpSystem_SecondaryHeatpumpGet_HeatpumpData_r_CompOutputTemp: 				st_Variable:= IotExtractType(monitor.Cooling.HeatPumpSystem.SecondaryHeatpumpGet.HeatpumpData.r_CompOutputTemp, 1, 0); 
// eDataMappingVarNames.Cooling_HeatPumpSystem_SecondaryHeatpumpGet_HeatpumpData_ui_WaterFlowRate: 				st_Variable:= IotExtractType(monitor.Cooling.HeatPumpSystem.SecondaryHeatpumpGet.HeatpumpData.ui_WaterFlowRate, 1, 0); 
// eDataMappingVarNames.Cooling_HeatPumpSystem_SecondaryHeatpumpGet_HeatpumpData_w_ErrorList_1: 				st_Variable:= IotExtractType(monitor.Cooling.HeatPumpSystem.SecondaryHeatpumpGet.HeatpumpData.w_ErrorList[1], 0, 0); 
// eDataMappingVarNames.Cooling_HeatPumpSystem_SecondaryHeatpumpGet_HeatpumpData_w_ErrorList_2: 				st_Variable:= IotExtractType(monitor.Cooling.HeatPumpSystem.SecondaryHeatpumpGet.HeatpumpData.w_ErrorList[2], 0, 0); 
// eDataMappingVarNames.Cooling_HeatPumpSystem_SecondaryHeatpumpGet_HeatpumpData_w_ErrorList_3: 				st_Variable:= IotExtractType(monitor.Cooling.HeatPumpSystem.SecondaryHeatpumpGet.HeatpumpData.w_ErrorList[3], 0, 0); 
// eDataMappingVarNames.Cooling_HeatPumpSystem_SecondaryHeatpumpGet_HeatpumpData_w_ErrorList_4: 				st_Variable:= IotExtractType(monitor.Cooling.HeatPumpSystem.SecondaryHeatpumpGet.HeatpumpData.w_ErrorList[4], 0, 0); 
// eDataMappingVarNames.Cooling_HeatPumpSystem_SecondaryHeatpumpGet_HeatpumpData_w_ErrorList_5: 				st_Variable:= IotExtractType(monitor.Cooling.HeatPumpSystem.SecondaryHeatpumpGet.HeatpumpData.w_ErrorList[5], 0, 0); 
// eDataMappingVarNames.Cooling_HeatPumpSystem_SecondaryHeatpumpGet_HeatpumpData_w_ErrorList_6: 				st_Variable:= IotExtractType(monitor.Cooling.HeatPumpSystem.SecondaryHeatpumpGet.HeatpumpData.w_ErrorList[6], 0, 0); 
// eDataMappingVarNames.Cooling_HeatPumpSystem_SecondaryHeatpumpGet_HeatpumpData_w_ErrorList_7: 				st_Variable:= IotExtractType(monitor.Cooling.HeatPumpSystem.SecondaryHeatpumpGet.HeatpumpData.w_ErrorList[7], 0, 0); 
// eDataMappingVarNames.Cooling_HeatPumpSystem_SecondaryHeatpumpGet_HeatpumpData_r_FanSpeedPCT: 				st_Variable:= IotExtractType(monitor.Cooling.HeatPumpSystem.SecondaryHeatpumpGet.HeatpumpData.r_FanSpeedPCT, 0, 0); 
// eDataMappingVarNames.Cooling_HeatPumpSystem_SecondaryHeatpumpGet_HeatpumpData_r_PumpSpeedPCT: 				st_Variable:= IotExtractType(monitor.Cooling.HeatPumpSystem.SecondaryHeatpumpGet.HeatpumpData.r_PumpSpeedPCT, 0, 0); 
// eDataMappingVarNames.Cooling_HeatPumpSystem_SecondaryHeatpumpGet_HeatpumpData_r_SetpointHeating: 				st_Variable:= IotExtractType(monitor.Cooling.HeatPumpSystem.SecondaryHeatpumpGet.HeatpumpData.r_SetpointHeating, 0, 0); 
// eDataMappingVarNames.Cooling_HeatPumpSystem_SecondaryHeatpumpGet_HeatpumpData_r_SetpointCooling: 				st_Variable:= IotExtractType(monitor.Cooling.HeatPumpSystem.SecondaryHeatpumpGet.HeatpumpData.r_SetpointCooling, 0, 0); 
// eDataMappingVarNames.Cooling_HeatPumpSystem_SecondaryHeatpumpGet_HeatpumpData_b_DefrostingActive: 				st_Variable:= IotExtractType(monitor.Cooling.HeatPumpSystem.SecondaryHeatpumpGet.HeatpumpData.b_DefrostingActive, 0, 0); 
// eDataMappingVarNames.Cooling_Events_b_SystemOvertemperatureWarning: 				st_Variable:= IotExtractType(monitor.Cooling.Events. .b_SystemOvertemperatureWarning, 0, 0); 
// eDataMappingVarNames.Cooling_Events_b_SystemUnderTemperatureWarning: 				st_Variable:= IotExtractType(monitor.Cooling.Events.b_SystemUnderTemperatureWarning, 0, 0); 
// eDataMappingVarNames.Cooling_Events_b_CoolingSystemFuseFailure: 				st_Variable:= IotExtractType(monitor.Cooling.Events.b_CoolingSystemFuseFailure, 0, 0); 
// eDataMappingVarNames.Cooling_Events_b_ACwaterPumpTimeOut: 				st_Variable:= IotExtractType(monitor.Cooling.Events.b_ACwaterPumpTimeOut, 0, 0); 
// eDataMappingVarNames.Cooling_Events_b_InverterLoopValveStuck: 				st_Variable:= IotExtractType(monitor.Cooling.Events.b_InverterLoopValveStuck, 0, 0); 
// eDataMappingVarNames.Cooling_Events_b_BattLoopValveStuck: 				st_Variable:= IotExtractType(monitor.Cooling.Events.b_BattLoopValveStuck, 0, 0); 
// eDataMappingVarNames.Cooling_Events_b_FancoilLoopValveStuck: 				st_Variable:= IotExtractType(monitor.Cooling.Events.b_FancoilLoopValveStuck, 0, 0); 
// eDataMappingVarNames.Cooling_Events_b_DCpumpPressureFault: 				st_Variable:= IotExtractType(monitor.Cooling.Events.b_DCpumpPressureFault, 0, 0); 
// eDataMappingVarNames.Cooling_Events_b_DCpumpTimeout: 				st_Variable:= IotExtractType(monitor.Cooling.Events.b_DCpumpTimeout, 0, 0); 
// eDataMappingVarNames.Cooling_Events_b_CoolingLoopIdlePressureWarning: 				st_Variable:= IotExtractType(monitor.Cooling.Events.b_CoolingLoopIdlePressureWarning, 0, 0); 
// eDataMappingVarNames.Cooling_Events_b_CoolingLoopIdlePressureError: 				st_Variable:= IotExtractType(monitor.Cooling.Events.b_CoolingLoopIdlePressureError, 0, 0); 
// eDataMappingVarNames.Cooling_Events_b_InverterCoolingLoopError: 				st_Variable:= IotExtractType(monitor.Cooling.Events.b_InverterCoolingLoopError, 0, 0); 
// eDataMappingVarNames.Cooling_Events_b_HeatpumpWarning: 				st_Variable:= IotExtractType(monitor.Cooling.Events.b_HeatpumpWarning, 0, 0); 
// eDataMappingVarNames.Cooling_Events_b_HeatPumpError: 				st_Variable:= IotExtractType(monitor.Cooling.Events.b_HeatPumpError, 0, 0); 
// eDataMappingVarNames.Cooling_Events_b_CoolantTempTooLow: 				st_Variable:= IotExtractType(monitor.Cooling.Events.b_CoolantTempTooLow, 0, 0); 
// eDataMappingVarNames.Cooling_Events_b_CoolantTempLow: 				st_Variable:= IotExtractType(monitor.Cooling.Events.b_CoolantTempLow, 0, 0); 
// eDataMappingVarNames.Cooling_Events_b_CoolantTempTooHigh: 				st_Variable:= IotExtractType(monitor.Cooling.Events.b_CoolantTempTooHigh, 0, 0); 
// eDataMappingVarNames.Cooling_Events_b_CoolantTempHigh: 				st_Variable:= IotExtractType(monitor.Cooling.Events.b_CoolantTempHigh, 0, 0); 
// eDataMappingVarNames.Router_Device_SystemUptime: 				st_Variable:= IotExtractType(monitor.Router.Device.SystemUptime, 0, 0); 
// eDataMappingVarNames.Router_Device_Temperature: 				st_Variable:= IotExtractType(monitor.Router.Device.Temperature, 0, 0); 
// eDataMappingVarNames.Router_Device_RouterSerial: 				st_Variable:= IotExtractType(monitor.Router.Device.RouterSerial, 0, 0); 
// eDataMappingVarNames.Router_GPS_Latitude: 				st_Variable:= IotExtractType(monitor.Router.GPS.Latitude, 0, 0); 
// eDataMappingVarNames.Router_GPS_Longitude: 				st_Variable:= IotExtractType(monitor.Router.GPS.Longitude, 0, 0); 
// eDataMappingVarNames.Router_GPS_FixTime: 				st_Variable:= IotExtractType(monitor.Router.GPS.FixTime, 0, 0); 
// eDataMappingVarNames.Router_GPS_DateTime: 				st_Variable:= IotExtractType(monitor.Router.GPS.DateTime, 0, 0); 
// eDataMappingVarNames.Router_GPS_Speed: 				st_Variable:= IotExtractType(monitor.Router.GPS.Speed, 0, 0); 
// eDataMappingVarNames.Router_GPS_SatCount: 				st_Variable:= IotExtractType(monitor.Router.GPS.SatCount, 0, 0); 
// eDataMappingVarNames.Router_GPS_Accuracy: 				st_Variable:= IotExtractType(monitor.Router.GPS.Accuracy, 0, 0); 
// eDataMappingVarNames.Router_Mobile_NetworkOperator: 				st_Variable:= IotExtractType(monitor.Router.Mobile.NetworkOperator, 0, 0); 
// eDataMappingVarNames.Router_Mobile_NetworkInfo: 				st_Variable:= IotExtractType(monitor.Router.Mobile.NetworkInfo, 0, 0); 
// eDataMappingVarNames.Router_Mobile_NetworkType: 				st_Variable:= IotExtractType(monitor.Router.Mobile.NetworkType, 0, 0); 
// eDataMappingVarNames.Router_Mobile_RSSI: 				st_Variable:= IotExtractType(monitor.Router.Mobile.RSSI, 0, 0); 
// eDataMappingVarNames.Router_Mobile_ui_Sim1DataSendMonth: 				st_Variable:= IotExtractType(monitor.Router.Mobile.ui_Sim1DataSendMonth, 0, 0); 
// eDataMappingVarNames.Router_Mobile_ui_Sim1DataReceivedMonth: 				st_Variable:= IotExtractType(monitor.Router.Mobile.ui_Sim1DataReceivedMonth, 0, 0); 
// eDataMappingVarNames.Router_Mobile_ui_Sim2DataSendMonth: 				st_Variable:= IotExtractType(monitor.Router.Mobile.ui_Sim2DataSendMonth, 0, 0); 
// eDataMappingVarNames.Router_Mobile_ui_Sim2DataReceivedMonth: 				st_Variable:= IotExtractType(monitor.Router.Mobile.ui_Sim2DataReceivedMonth, 0, 0); 
// eDataMappingVarNames.Router_Mobile_s_EmergencySMSNumber: 				st_Variable:= IotExtractType(monitor.Router.Mobile.s_EmergencySMSNumber, 0, 0); 
// eDataMappingVarNames.Router_Mobile_s_SecondarySMSNumber: 				st_Variable:= IotExtractType(monitor.Router.Mobile.s_SecondarySMSNumber, 0, 0); 
// eDataMappingVarNames.Router_Mobile_s_EmergencySMSDevName: 				st_Variable:= IotExtractType(monitor.Router.Mobile.s_EmergencySMSDevName, 0, 0); 
// eDataMappingVarNames.Router_Mobile_st_LatestSMSMessage: 				st_Variable:= IotExtractType(monitor.Router.Mobile.st_LatestSMSMessage, 0, 0); 
